# B&R Automation Studio project NAELD004C00R10L518F00 (part 15)

#### Act_OptP0937FBCtrl.st
```iecst
ACTION Act_OptP0937FBCtrl:

	fbJogSlowToFastDlyTm.PT			:= T#2s;
	fbJogSlowToFastDlyTm;
	fbLmtRstTm;

	//Conveyor Sensor Interruption
	IF p_tyDI.bPullerRetRS = FALSE AND eCurrPage = UIP0937AWPushOrPuller THEN
		tyP0937AWPushOrPuller.tyMotionStd.tyBtnStop.bRtCompl	:= TRUE;
	END_IF

//	IF EDGEPOS((p_udiAWPushOrPullerAxisErrID = 21570 OR p_udiAWPushOrPullerAxisErrID = 21571)
	IF EDGEPOS ((p_bAWPushOrPullerFwdLmtSen OR p_bAWPushOrPullerRevLmtSen)
		AND tyP0937AWPushOrPuller.tyMotionStd.tyBtnJogOpen.bValue = FALSE
		AND tyP0937AWPushOrPuller.tyMotionStd.tyBtnJogClose.bValue = FALSE)
	THEN
		fbLmtRstTm.IN	:= TRUE;
	END_IF

	IF fbLmtRstTm.Q = TRUE THEN
		tyP0937AWPushOrPuller.tyMotionStd.tyBtnRst.bRtCompl		:= TRUE;
	END_IF

	IF (tyP0937AWPushOrPuller.tyMotionStd.tyBtnJogOpen.bValue = FALSE AND tyP0937AWPushOrPuller.tyMotionStd.tyBtnJogClose.bValue = FALSE) AND (p_bAWPushOrPullerJogging = TRUE) THEN
		bJogStopAWPushOrPuller	:= TRUE;
	END_IF

	IF tyP0937AWPushOrPuller.tyMotionStd.tyBtnStop.bRtCompl = TRUE THEN
		eAWPushOrPullerAct		:= AWActStop;

		IF p_eAWPushOrPullerStat = AWActStop AND p_eAWPushOrPullerStatus = Done THEN
			eAWPushOrPullerAct	:= AWActIdle;

			tyP0937AWPushOrPuller.tyMotionStd.tyBtnStop.bRtCompl	:= FALSE;
			tyP0937AWPushOrPuller.tyMotionStd.tyBtnJogOpen.bRtCompl	:= FALSE;
			tyP0937AWPushOrPuller.tyMotionStd.tyBtnJogClose.bRtCompl:= FALSE;
			tyP0937AWPushOrPuller.tyMotionStd.tyBtnOrigin.bRtCompl	:= FALSE;
			tyP0937AWPushOrPuller.tyMotionStd.tyBtnMovAbs.bRtCompl	:= FALSE;
			tyP0937AWPushOrPuller.tyMotionStd.tyBtnMovRel.bRtCompl	:= FALSE;
			tyP0937AWPushOrPuller.tyAW.tyBtnGo.bRtCompl				:= FALSE;

			tyP0937AWPushOrPuller.tyMotionStd.tyBtnStop.bValue		:= TRUE;
			tyP0937AWPushOrPuller.tyMotionStd.tyBtnJogOpen.bValue	:= FALSE;
			tyP0937AWPushOrPuller.tyMotionStd.tyBtnJogClose.bValue	:= FALSE;
			tyP0937AWPushOrPuller.tyMotionStd.tyBtnOrigin.bValue	:= FALSE;
			tyP0937AWPushOrPuller.tyMotionStd.tyBtnMovAbs.bValue	:= FALSE;
			tyP0937AWPushOrPuller.tyMotionStd.tyBtnMovRel.bValue	:= FALSE;
			tyP0937AWPushOrPuller.tyAW.tyBtnGo.bValue				:= FALSE;

			tyP0937AWPushOrPuller.tyMotionStd.tyBtnStop.bRtLk		:= TRUE;
			tyP0937AWPushOrPuller.tyMotionStd.tyBtnJogOpen.bRtLk	:= FALSE;
			tyP0937AWPushOrPuller.tyMotionStd.tyBtnJogClose.bRtLk	:= FALSE;
			tyP0937AWPushOrPuller.tyMotionStd.tyBtnOrigin.bRtLk		:= FALSE;
			tyP0937AWPushOrPuller.tyMotionStd.tyBtnMovAbs.bRtLk		:= FALSE;
			tyP0937AWPushOrPuller.tyMotionStd.tyBtnMovRel.bRtLk		:= FALSE;
			tyP0937AWPushOrPuller.tyAW.tyBtnGo.bRtLk				:= FALSE;
		END_IF

	ELSIF (tyP0937AWPushOrPuller.tyMotionStd.tyBtnJogOpen.bRtCompl = TRUE) OR (tyP0937AWPushOrPuller.tyMotionStd.tyBtnJogClose.bRtCompl = TRUE) OR (bJogStopAWPushOrPuller = TRUE) THEN
		bJogSlow					:= FALSE;
		bJogFast					:= FALSE;
		fbJogSlowToFastDlyTm.IN		:= FALSE;

		eAWPushOrPullerAct		:= AWActJogStop;

		IF p_eAWPushOrPullerStat = AWActJogStop AND p_eAWPushOrPullerStatus = Done THEN
			eAWPushOrPullerAct	:= AWActIdle;

			bJogStopAWPushOrPuller	:= FALSE;

			tyP0937AWPushOrPuller.tyMotionStd.tyBtnStop.bRtCompl	:= FALSE;
			tyP0937AWPushOrPuller.tyMotionStd.tyBtnJogOpen.bRtCompl	:= FALSE;
			tyP0937AWPushOrPuller.tyMotionStd.tyBtnJogClose.bRtCompl:= FALSE;
			tyP0937AWPushOrPuller.tyMotionStd.tyBtnOrigin.bRtCompl	:= FALSE;
			tyP0937AWPushOrPuller.tyMotionStd.tyBtnMovAbs.bRtCompl	:= FALSE;
			tyP0937AWPushOrPuller.tyMotionStd.tyBtnMovRel.bRtCompl	:= FALSE;
			tyP0937AWPushOrPuller.tyAW.tyBtnGo.bRtCompl				:= FALSE;

			tyP0937AWPushOrPuller.tyMotionStd.tyBtnStop.bValue		:= TRUE;
			tyP0937AWPushOrPuller.tyMotionStd.tyBtnJogOpen.bValue	:= FALSE;
			tyP0937AWPushOrPuller.tyMotionStd.tyBtnJogClose.bValue	:= FALSE;
			tyP0937AWPushOrPuller.tyMotionStd.tyBtnOrigin.bValue	:= FALSE;
			tyP0937AWPushOrPuller.tyMotionStd.tyBtnMovAbs.bValue	:= FALSE;
			tyP0937AWPushOrPuller.tyMotionStd.tyBtnMovRel.bValue	:= FALSE;
			tyP0937AWPushOrPuller.tyAW.tyBtnGo.bValue				:= FALSE;

			tyP0937AWPushOrPuller.tyMotionStd.tyBtnStop.bRtLk		:= TRUE;
			tyP0937AWPushOrPuller.tyMotionStd.tyBtnJogOpen.bRtLk	:= FALSE;
			tyP0937AWPushOrPuller.tyMotionStd.tyBtnJogClose.bRtLk	:= FALSE;
			tyP0937AWPushOrPuller.tyMotionStd.tyBtnOrigin.bRtLk		:= FALSE;
			tyP0937AWPushOrPuller.tyMotionStd.tyBtnMovAbs.bRtLk		:= FALSE;
			tyP0937AWPushOrPuller.tyMotionStd.tyBtnMovRel.bRtLk		:= FALSE;
			tyP0937AWPushOrPuller.tyAW.tyBtnGo.bRtLk				:= FALSE;
		END_IF

	ELSIF tyP0937AWPushOrPuller.tyMotionStd.tyBtnPwr.bRtCompl = TRUE THEN
		tyP0937AWPushOrPuller.tyMotionStd.tyBtnPwr.bRtLk	:= TRUE;

		IF tyP0937AWPushOrPuller.tyMotionStd.tyBtnPwr.bValue = TRUE THEN
			eAWPushOrPullerAct		:= AWActPwrOn;

			IF p_eAWPushOrPullerStat = AWActPwrOn AND p_eAWPushOrPullerStatus = Done THEN
				eAWPushOrPullerAct	:= AWActIdle;

				tyP0937AWPushOrPuller.tyMotionStd.tyBtnPwr.bRtCompl	:= FALSE;
				tyP0937AWPushOrPuller.tyMotionStd.tyBtnPwr.bRtLk		:= FALSE;
			END_IF
		ELSE
			eAWPushOrPullerAct	:= AWActPwrOff;

			IF p_eAWPushOrPullerStat = AWActPwrOff AND p_eAWPushOrPullerStatus = Done THEN
				eAWPushOrPullerAct	:= AWActIdle;

				tyP0937AWPushOrPuller.tyMotionStd.tyBtnPwr.bRtCompl			:= FALSE;
				tyP0937AWPushOrPuller.tyMotionStd.tyBtnPwr.bRtLk			:= FALSE;
			END_IF
		END_IF

	ELSIF tyP0937AWPushOrPuller.tyMotionStd.tyBtnOrigin.bRtCompl = TRUE THEN
		tyP0937AWPushOrPuller.tyMotionStd.tyBtnOrigin.bValue	:= TRUE;
		tyP0937AWPushOrPuller.tyMotionStd.tyBtnStop.bValue	:= FALSE;

		tyP0937AWPushOrPuller.tyMotionStd.tyBtnOrigin.bRtLk	:= TRUE;
		tyP0937AWPushOrPuller.tyMotionStd.tyBtnStop.bRtLk		:= FALSE;

		eAWPushOrPullerAct		:= AWActHoming;

		IF p_eAWPushOrPullerStat = AWActHoming AND p_eAWPushOrPullerStatus = Done THEN
			eAWPushOrPullerAct	:= AWActIdle;

			tyP0937AWPushOrPuller.tyMotionStd.tyBtnOrigin.bRtCompl	:= FALSE;
			tyP0937AWPushOrPuller.tyMotionStd.tyBtnOrigin.bValue		:= FALSE;
			tyP0937AWPushOrPuller.tyMotionStd.tyBtnStop.bValue		:= TRUE;

			tyP0937AWPushOrPuller.tyMotionStd.tyBtnOrigin.bRtLk		:= FALSE;
			tyP0937AWPushOrPuller.tyMotionStd.tyBtnStop.bRtLk			:= TRUE;
		END_IF

	ELSIF tyP0937AWPushOrPuller.tyMotionStd.tyBtnRst.bRtCompl = TRUE THEN
		tyP0937AWPushOrPuller.tyMotionStd.tyBtnRst.bValue					:= TRUE;
		tyP0937AWPushOrPuller.tyMotionStd.tyBtnRst.bRtLk					:= TRUE;

		eAWPushOrPullerAct		:= AWActRstAxisErr;

		IF p_eAWPushOrPullerStat = AWActRstAxisErr AND p_eAWPushOrPullerStatus = Done THEN
			eAWPushOrPullerAct	:= AWActIdle;

			tyP0937AWPushOrPuller.tyMotionStd.tyBtnRst.bRtCompl		:= FALSE;
			tyP0937AWPushOrPuller.tyMotionStd.tyBtnRst.bValue			:= FALSE;
			tyP0937AWPushOrPuller.tyMotionStd.tyBtnRst.bRtLk			:= FALSE;

			fbLmtRstTm.IN			:= FALSE;
		END_IF

	ELSIF tyP0937AWPushOrPuller.tyAW.tyBtnGo.bRtCompl = TRUE THEN
		tyP0937AWPushOrPuller.tyAW.tyBtnGo.bValue				:= TRUE;
		tyP0937AWPushOrPuller.tyMotionStd.tyBtnStop.bValue	:= FALSE;

		tyP0937AWPushOrPuller.tyAW.tyBtnGo.bRtLk				:= TRUE;
		tyP0937AWPushOrPuller.tyMotionStd.tyBtnStop.bRtLk		:= FALSE;

		diMnlAWPushOrPullerGoWidth	:= (tyP0937AWPushOrPuller.tyAW.tyNumNewWidth.diValue)*3/4;
		diMnlAWPushOrPullerNomSpd		:= tyP0937AWPushOrPuller.tyMotionStd.tyNumNomSpd.diValue;

		eAWPushOrPullerAct		:= AWActGoWidth;

		IF p_eAWPushOrPullerStat = AWActGoWidth AND p_eAWPushOrPullerStatus = Done THEN
			eAWPushOrPullerAct	:= AWActIdle;

			tyP0937AWPushOrPuller.tyAW.tyBtnGo.bRtCompl			:= FALSE;
			tyP0937AWPushOrPuller.tyAW.tyBtnGo.bValue				:= FALSE;
			tyP0937AWPushOrPuller.tyMotionStd.tyBtnStop.bValue	:= TRUE;

			tyP0937AWPushOrPuller.tyAW.tyBtnGo.bRtLk				:= FALSE;
			tyP0937AWPushOrPuller.tyMotionStd.tyBtnStop.bRtLk		:= TRUE;
		END_IF

	ELSIF tyP0937AWPushOrPuller.tyMotionStd.tyBtnMovAbs.bRtCompl = TRUE THEN
		tyP0937AWPushOrPuller.tyMotionStd.tyBtnMovAbs.bValue		:= TRUE;
		tyP0937AWPushOrPuller.tyMotionStd.tyBtnStop.bValue		:= FALSE;

		tyP0937AWPushOrPuller.tyMotionStd.tyBtnMovAbs.bRtLk		:= TRUE;
		tyP0937AWPushOrPuller.tyMotionStd.tyBtnStop.bRtLk			:= FALSE;

		diMnlAWPushOrPullerTargetPos	:= tyP0937AWPushOrPuller.tyMotionStd.tyNumTargetPos.diValue;
		diMnlAWPushOrPullerNomSpd		:= tyP0937AWPushOrPuller.tyMotionStd.tyNumNomSpd.diValue;

		eAWPushOrPullerAct		:= AWActMovAbs;

		IF p_eAWPushOrPullerStat = AWActMovAbs AND p_eAWPushOrPullerStatus = Done THEN
			eAWPushOrPullerAct	:= AWActIdle;

			tyP0937AWPushOrPuller.tyMotionStd.tyBtnMovAbs.bRtCompl	:= FALSE;
			tyP0937AWPushOrPuller.tyMotionStd.tyBtnMovAbs.bValue		:= FALSE;
			tyP0937AWPushOrPuller.tyMotionStd.tyBtnStop.bValue		:= TRUE;

			tyP0937AWPushOrPuller.tyMotionStd.tyBtnMovAbs.bRtLk		:= FALSE;
			tyP0937AWPushOrPuller.tyMotionStd.tyBtnStop.bRtLk			:= TRUE;
		END_IF

	ELSIF tyP0937AWPushOrPuller.tyMotionStd.tyBtnMovRel.bRtCompl = TRUE THEN
		tyP0937AWPushOrPuller.tyMotionStd.tyBtnMovRel.bValue			:= TRUE;
		tyP0937AWPushOrPuller.tyMotionStd.tyBtnStop.bValue			:= FALSE;

		tyP0937AWPushOrPuller.tyMotionStd.tyBtnMovRel.bRtLk			:= TRUE;
		tyP0937AWPushOrPuller.tyMotionStd.tyBtnStop.bRtLk				:= FALSE;

		diMnlAWPushOrPullerStepSize	:= tyP0937AWPushOrPuller.tyMotionStd.tyNumStepSize.diValue;
		diMnlAWPushOrPullerNomSpd		:= tyP0937AWPushOrPuller.tyMotionStd.tyNumNomSpd.diValue;

		eAWPushOrPullerAct		:= AWActMovRel;

		IF p_eAWPushOrPullerStat = AWActMovRel AND p_eAWPushOrPullerStatus = Done THEN
			eAWPushOrPullerAct	:= AWActIdle;

			tyP0937AWPushOrPuller.tyMotionStd.tyBtnMovRel.bRtCompl	:= FALSE;
			tyP0937AWPushOrPuller.tyMotionStd.tyBtnMovRel.bValue		:= FALSE;
			tyP0937AWPushOrPuller.tyMotionStd.tyBtnStop.bValue		:= TRUE;

			tyP0937AWPushOrPuller.tyMotionStd.tyBtnMovRel.bRtLk		:= FALSE;
			tyP0937AWPushOrPuller.tyMotionStd.tyBtnStop.bRtLk			:= TRUE;
		END_IF

	ELSIF (tyP0937AWPushOrPuller.tyMotionStd.tyBtnJogOpen.bValue = TRUE) AND (fbJogSlowToFastDlyTm.Q = FALSE) AND (bJogSlow = FALSE) THEN
		tyP0937AWPushOrPuller.tyMotionStd.tyBtnStop.bValue		:= FALSE;
		tyP0937AWPushOrPuller.tyMotionStd.tyBtnStop.bRtLk			:= FALSE;

		fbJogSlowToFastDlyTm.IN	:= TRUE;

		diMnlAWPushOrPullerJogSpd		:= tyP0937AWPushOrPuller.tyMotionStd.tyNumSlwSpd.diValue;

		eAWPushOrPullerAct		:= AWActJogOpen;

		IF p_eAWPushOrPullerStat = AWActJogOpen AND p_eAWPushOrPullerStatus = Done THEN
			eAWPushOrPullerAct	:= AWActIdle;
			bJogSlow		:= TRUE;
		ELSIF p_eAWPushOrPullerStatus = Error THEN
			fbJogSlowToFastDlyTm.IN	:= FALSE;
			bJogSlow		:= TRUE;
		END_IF

	ELSIF (tyP0937AWPushOrPuller.tyMotionStd.tyBtnJogOpen.bValue = TRUE) AND (fbJogSlowToFastDlyTm.Q = TRUE) AND (bJogFast = FALSE) THEN
		tyP0937AWPushOrPuller.tyMotionStd.tyBtnStop.bValue	:= FALSE;
		tyP0937AWPushOrPuller.tyMotionStd.tyBtnStop.bRtLk		:= FALSE;

		fbJogSlowToFastDlyTm.IN		:= TRUE;

		diMnlAWPushOrPullerJogSpd		:= tyP0937AWPushOrPuller.tyMotionStd.tyNumNomSpd.diValue;

		eAWPushOrPullerAct	:= AWActJogOpen;

		IF p_eAWPushOrPullerStat = AWActJogOpen AND p_eAWPushOrPullerStatus = Done THEN
			eAWPushOrPullerAct	:= AWActIdle;
			bJogFast				:= TRUE;
		ELSIF p_eAWPushOrPullerStatus = Error THEN
			fbJogSlowToFastDlyTm.IN	:= FALSE;
			bJogFast				:= TRUE;
		END_IF

	ELSIF (tyP0937AWPushOrPuller.tyMotionStd.tyBtnJogClose.bValue = TRUE) AND (fbJogSlowToFastDlyTm.Q = FALSE) AND (bJogSlow = FALSE) THEN
		tyP0937AWPushOrPuller.tyMotionStd.tyBtnStop.bValue					:= FALSE;
		tyP0937AWPushOrPuller.tyMotionStd.tyBtnStop.bRtLk					:= FALSE;

		fbJogSlowToFastDlyTm.IN		:= TRUE;

		diMnlAWPushOrPullerJogSpd		:= tyP0937AWPushOrPuller.tyMotionStd.tyNumSlwSpd.diValue;

		eAWPushOrPullerAct		:= AWActJogClose;

		IF p_eAWPushOrPullerStat = AWActJogClose AND p_eAWPushOrPullerStatus = Done THEN
			eAWPushOrPullerAct	:= AWActIdle;
			bJogSlow				:= TRUE;
		ELSIF p_eAWPushOrPullerStatus = Error THEN
			fbJogSlowToFastDlyTm.IN	:= FALSE;
			bJogSlow				:= TRUE;
		END_IF

	ELSIF (tyP0937AWPushOrPuller.tyMotionStd.tyBtnJogClose.bValue = TRUE) AND (fbJogSlowToFastDlyTm.Q = TRUE) AND (bJogFast = FALSE) THEN
		tyP0937AWPushOrPuller.tyMotionStd.tyBtnStop.bValue	:= FALSE;
		tyP0937AWPushOrPuller.tyMotionStd.tyBtnStop.bRtLk		:= FALSE;

		fbJogSlowToFastDlyTm.IN		:= TRUE;

		diMnlAWPushOrPullerJogSpd		:= tyP0937AWPushOrPuller.tyMotionStd.tyNumNomSpd.diValue;

		eAWPushOrPullerAct			:= AWActJogClose;

		IF p_eAWPushOrPullerStat = AWActJogClose AND p_eAWPushOrPullerStatus = Done THEN
			eAWPushOrPullerAct	:= AWActIdle;
			bJogFast				:= TRUE;
		ELSIF p_eAWPushOrPullerStatus = Error THEN
			fbJogSlowToFastDlyTm.IN	:= FALSE;
			bJogFast				:= TRUE;
		END_IF

	END_IF

END_ACTION
```

#### Act_OptP0937FullMask.st
```iecst
ACTION Act_OptP0937FullMask:

	IF eCurrPage = UIP0937AWPushOrPuller THEN

		IF p_tyDI.bEStopSig = FALSE THEN
			p_tyC0002FullMask ACCESS ADR(tyP0937AWPushOrPuller.tyFullMaskEStop);

		ELSIF p_tyDI.bCoverSWSig = FALSE THEN
			p_tyC0002FullMask ACCESS ADR(tyP0937AWPushOrPuller.tyFullMaskCWSig);

		ELSIF p_tyDI.bSafetyRlySig = FALSE THEN
			p_tyC0002FullMask ACCESS ADR(tyP0937AWPushOrPuller.tyFullMaskSafetyRly);

		ELSIF p_tyDI.bConvLftSen THEN
			p_tyC0002FullMask ACCESS ADR(tyP0937AWPushOrPuller.tyFullMaskLftSenInterrupt);

		ELSIF p_tyDI.bConvRgtSen THEN
			p_tyC0002FullMask ACCESS ADR(tyP0937AWPushOrPuller.tyFullMaskRgtSenInterrupt);

		ELSIF p_tyNtParamCurr.bProjInletShutPrep AND (p_tyDI.bInShutterCloseRS = FALSE
			OR (p_tyDI.bInShutterCloseRS2 = FALSE AND p_tyNtParamCurr.tyDISettings.diInShutterCloseRS2 > 0)
			OR (p_tyDI.bInShutterCloseRS3 = FALSE AND p_tyNtParamCurr.tyDISettings.diInShutterCloseRS3 > 0)) THEN
			IF p_tyNtParamCurr.bProjCurtainSenPrep THEN
				IF p_tyDI.bInShutterCloseRS = FALSE OR p_tyDI.bInShutterCloseRS2 = FALSE OR p_tyDI.bInShutterCloseRS3 = FALSE THEN
					p_tyC0002FullMask ACCESS ADR(tyP0937AWPushOrPuller.tyFullMaskInShutOpnInterrupt);
				END_IF
			ELSE
				IF p_tyDI.bInShutterCloseRS = FALSE THEN
					p_tyC0002FullMask ACCESS ADR(tyP0937AWPushOrPuller.tyFullMaskInShutOpnInterrupt);
				END_IF
			END_IF

	//	ELSIF p_tyNtParamCurr.bProjOutletShutPrep AND p_tyDI.bOutShutterCloseRS = FALSE AND p_McParamOutShutterDis = FALSE THEN
		ELSIF p_tyNtParamCurr.bProjOutletShutPrep AND p_tyDI.bOutShutterCloseRS = FALSE THEN
			p_tyC0002FullMask ACCESS ADR(tyP0937AWPushOrPuller.tyFullMaskOutShutOpnInterrupt);

		ELSIF  p_tyDI.bPullerRetRS = FALSE OR p_tyDI.bPullerRotHmRS = FALSE THEN
			p_tyC0002FullMask ACCESS ADR(tyP0937AWPushOrPuller.tyFullMaskPullerRetInterrupt);

		ELSE
			p_tyC0002FullMask ACCESS ADR(tyP0937AWPushOrPuller.tyFullMaskHide);

		END_IF

	END_IF

END_ACTION
```

#### Act_OptP0937UpdtDat.st
```iecst
ACTION Act_OptP0937UpdtDat:

	tyP0937AWPushOrPuller.tyMotionStd.tyNumCurrPos.diValue		:= p_diAWPushOrPullerActualPos;
	tyP0937AWPushOrPuller.tyMotionStd.tyNumErrCode.diValue		:= UDINT_TO_DINT(p_udiAWPushOrPullerAxisErrID);
	tyP0937AWPushOrPuller.tyMotionStd.tyBitmapPwr.usiValueIdx		:= BOOL_TO_USINT(p_bAWPushOrPullerPwrOn);
	tyP0937AWPushOrPuller.tyMotionStd.tyBitmapRst.usiValueIdx		:= BOOL_TO_USINT(NOT p_bAWPushOrPullerAxisErr);
	tyP0937AWPushOrPuller.tyMotionStd.tyBitmapOrigin.usiValueIdx	:= BOOL_TO_USINT(p_bAWPushOrPullerIsHomed);
	tyP0937AWPushOrPuller.tyMotionStd.tyBtnOpenLmtSen.bValue		:= p_bAWPushOrPullerCloseSen;
	tyP0937AWPushOrPuller.tyMotionStd.tyBtnCloseLmtSen.bValue		:= p_bAWPushOrPullerOpenSen;

	IF p_bAWPushOrPullerIsHomed = TRUE THEN
		IF p_diAWPushOrPullerActualPos <= (p_tyNtParamCurr.tyProdRcpWidth.diMax / 2) THEN
			tyP0937AWPushOrPuller.tyMotionStd.tyBitmapMc.uiValueIdx 	:= 38;
		ELSE
			tyP0937AWPushOrPuller.tyMotionStd.tyBitmapMc.uiValueIdx 	:= 39;
		END_IF
	ELSE
		tyP0937AWPushOrPuller.tyMotionStd.tyBitmapMc.uiValueIdx	:= 38;
	END_IF

	IF p_tyNtParamCurr.eProjMag = LDMagTriple AND p_tyNtParamCurr.bMagAutoVerifyPrep = FALSE AND p_tyNtParamCurr.bProjMotorizedPullerPrep = TRUE
		AND p_tyNtParamCurr.bProjCurtainSenPrep = FALSE THEN
		IF 	tyP0937AWPushOrPuller.tyMotionStd.tyBitmapMc.uiValueIdx < 300 THEN
			tyP0937AWPushOrPuller.tyMotionStd.tyBitmapMc.uiValueIdx	:= tyP0937AWPushOrPuller.tyMotionStd.tyBitmapMc.uiValueIdx + 300;
		END_IF
	ELSIF p_tyNtParamCurr.eProjMag = LDMagTriple AND p_tyNtParamCurr.bMagAutoVerifyPrep = FALSE AND p_tyNtParamCurr.bProjMotorizedPullerPrep = TRUE
		AND p_tyNtParamCurr.bProjCurtainSenPrep = TRUE AND p_tyNtParamCurr.bProjTopToBtmDefault = TRUE THEN
		IF 	tyP0937AWPushOrPuller.tyMotionStd.tyBitmapMc.uiValueIdx < 373-38 THEN
			tyP0937AWPushOrPuller.tyMotionStd.tyBitmapMc.uiValueIdx	:= tyP0937AWPushOrPuller.tyMotionStd.tyBitmapMc.uiValueIdx + 373-38;
		END_IF
	ELSIF p_tyNtParamCurr.eProjMag = LDMagTriple AND p_tyNtParamCurr.bMagAutoVerifyPrep = FALSE AND p_tyNtParamCurr.bProjMotorizedPullerPrep = TRUE
		AND p_tyNtParamCurr.bProjCurtainSenPrep = TRUE AND p_tyNtParamCurr.bProjTopToBtmDefault = FALSE THEN
		IF 	tyP0937AWPushOrPuller.tyMotionStd.tyBitmapMc.uiValueIdx < 428-38 THEN
			tyP0937AWPushOrPuller.tyMotionStd.tyBitmapMc.uiValueIdx	:= tyP0937AWPushOrPuller.tyMotionStd.tyBitmapMc.uiValueIdx + 428-38;

		END_IF
	END_IF

END_ACTION
```

#### Act_EntP0939Disp.st
```iecst
ACTION Act_EntP0939Disp:

	//Access Address
	p_tyC0002FullMask ACCESS ADR(tyP0939MagConv4.tyFullMaskHide);

//	p_tyC0004Navi ACCESS ADR(tyP0939MagConv4.tyNaviBack);
	p_tyC0004Navi ACCESS ADR(tyP0939MagConv4.tyNavi4Lyr4);

	p_tyC0005Main ACCESS ADR(tyCommon.tyMain);

	p_tyC0007Notif ACCESS ADR(tyCommon.tyNotif);

	p_tyC0008MsgBox ACCESS ADR(tyP0939MagConv4.tyMsgBoxHide);

	p_tyC0009Info ACCESS ADR(tyCommon.tyInfo);

	p_tyP0939Mag4ConvCom ACCESS ADR(tyP0939MagConv4.tyCom);
	p_tyP0939Mag4ConvDC ACCESS ADR(tyP0939MagConv4.tyDC);
	p_tyP0939Mag4ConvFB ACCESS ADR(tyP0939MagConv4.tyFB);

	IF p_tyNtParamCurr.eProjMag = LDMagDual AND p_tyNtParamCurr.bMagAutoVerifyPrep = FALSE THEN
		tyP0939MagConv4.tyCom.tyBitmapMc.usiValueIdx	:= 111;
	ELSIF p_tyNtParamCurr.eProjMag = LDMagDual AND p_tyNtParamCurr.bMagAutoVerifyPrep = TRUE THEN
		tyP0939MagConv4.tyCom.tyBitmapMc.usiValueIdx	:= 200;
	ELSIF p_tyNtParamCurr.eProjMag = LDMagTriple AND p_tyNtParamCurr.bMagAutoVerifyPrep = TRUE THEN
		tyP0939MagConv4.tyCom.tyBitmapMc.usiValueIdx	:= 0;
	ELSIF p_tyNtParamCurr.eProjMag = LDMagQuadruple AND p_tyNtParamCurr.bMagAutoVerifyPrep = TRUE THEN
		tyP0939MagConv4.tyCom.tyBitmapMc.usiValueIdx	:= 116;
	ELSE
		tyP0939MagConv4.tyCom.tyBitmapMc.usiValueIdx	:= 100;
	END_IF

	IF p_tyNtParamCurr.bMagAutoVerifyPrep = FALSE THEN
		tyP0939MagConv4.tyFB.tyBtnFixedClamp.usiTxtIdx	:= 6;
		tyP0939MagConv4.tyFB.tyBtnFixedUnclamp.usiTxtIdx:= 6;
		tyP0939MagConv4.tyFB.tyBtnRemoteClamp.usiTxtIdx	:= 6;
		tyP0939MagConv4.tyFB.tyBtnRemoteUnclamp.usiTxtIdx:= 6;
	ELSE
		tyP0939MagConv4.tyFB.tyBtnFixedClamp.usiTxtIdx	:= 6;
		tyP0939MagConv4.tyFB.tyBtnFixedUnclamp.usiTxtIdx:= 6;
		tyP0939MagConv4.tyFB.tyBtnRemoteClamp.usiTxtIdx	:= 6;
		tyP0939MagConv4.tyFB.tyBtnRemoteUnclamp.usiTxtIdx:= 6;

	END_IF

	IF p_tyNtParamCurr.bMagAutoVerifyPrep = FALSE THEN
		IF tyP0939MagConv4.tyCom.tyBtnSwitch.bValue THEN
			fUIInRtStatHide(ADR(tyP0939MagConv4.tyFB.tyLyr.uiRtStat));
			fUIInRtStatHide(ADR(tyP0939MagConv4.tyDC.tyLyr.uiRtStat));
			fUIInRtStatHide(ADR(tyP0939MagConv4.tyFB.tyLyrWithoutSelClamp.uiRtStat));
			fUIInRtStatOff(ADR(tyP0939MagConv4.tyDC.tyLyrWithoutSelClamp.uiRtStat));
		ELSE
			fUIInRtStatHide(ADR(tyP0939MagConv4.tyFB.tyLyr.uiRtStat));
			fUIInRtStatHide(ADR(tyP0939MagConv4.tyDC.tyLyr.uiRtStat));
			fUIInRtStatOff(ADR(tyP0939MagConv4.tyFB.tyLyrWithoutSelClamp.uiRtStat));
			fUIInRtStatHide(ADR(tyP0939MagConv4.tyDC.tyLyrWithoutSelClamp.uiRtStat));
		END_IF
	ELSE
		IF tyP0939MagConv4.tyCom.tyBtnSwitch.bValue THEN
			fUIInRtStatHide(ADR(tyP0939MagConv4.tyFB.tyLyr.uiRtStat));
			fUIInRtStatOff(ADR(tyP0939MagConv4.tyDC.tyLyr.uiRtStat));
			fUIInRtStatHide(ADR(tyP0939MagConv4.tyFB.tyLyrWithoutSelClamp.uiRtStat));
			fUIInRtStatHide(ADR(tyP0939MagConv4.tyDC.tyLyrWithoutSelClamp.uiRtStat));
		ELSE
			fUIInRtStatOff(ADR(tyP0939MagConv4.tyFB.tyLyr.uiRtStat));
			fUIInRtStatHide(ADR(tyP0939MagConv4.tyDC.tyLyr.uiRtStat));
			fUIInRtStatHide(ADR(tyP0939MagConv4.tyFB.tyLyrWithoutSelClamp.uiRtStat));
			fUIInRtStatHide(ADR(tyP0939MagConv4.tyDC.tyLyrWithoutSelClamp.uiRtStat));
		END_IF
	END_IF

END_ACTION
```

#### Act_OptP0939FullMask.st
```iecst
ACTION Act_OptP0939FullMask:

	IF eCurrPage = UIP0939MagConv4 THEN

		IF p_tyDI.bEStopSig = FALSE THEN
			p_tyC0002FullMask ACCESS ADR(tyP0939MagConv4.tyFullMaskEStop);

		ELSIF p_tyDI.bCoverSWSig = FALSE THEN
			p_tyC0002FullMask ACCESS ADR(tyP0939MagConv4.tyFullMaskCWSig);

		ELSIF p_tyDI.bSafetyRlySig = FALSE THEN
			p_tyC0002FullMask ACCESS ADR(tyP0939MagConv4.tyFullMaskSafetyRly);

		ELSE
			p_tyC0002FullMask ACCESS ADR(tyP0939MagConv4.tyFullMaskHide);

		END_IF

	END_IF

END_ACTION
```

#### Act_OptP0939Navi.st
```iecst
ACTION Act_OptP0939Navi:

	IF tyP0939MagConv4.tyNavi4Lyr4.tyBtnBack.bRtCompl = TRUE THEN
		tyP0939MagConv4.tyNavi4Lyr4.tyBtnBack.bRtCompl	:= FALSE;
		tyP0939MagConv4.tyNavi4Lyr4.tyBtnBack.bValue	:= FALSE;

		eChgPage	:= UIP0920MtrNPneuCtrl;

		bDispMagConv1	:= FALSE;
		bDispMagConv2	:= FALSE;
		bDispMagConv3	:= FALSE;
		bDispMagConv4	:= TRUE;

	ELSIF tyP0939MagConv4.tyNavi4Lyr4.tyBtnLeft.bRtCompl = TRUE THEN
		tyP0939MagConv4.tyNavi4Lyr4.tyBtnLeft.bRtCompl			:= FALSE;
		tyP0939MagConv4.tyNavi4Lyr4.tyBtnLeft.bValue			:= FALSE;
		eChgPage												:= UIP0932MagConv3;
		bDispMagConv1	:= FALSE;
		bDispMagConv2	:= FALSE;
		bDispMagConv3	:= TRUE;
		bDispMagConv4	:= FALSE;

	ELSIF tyP0939MagConv4.tyNavi4Lyr4.tyBtnRgt.bRtCompl = TRUE THEN
		tyP0939MagConv4.tyNavi4Lyr4.tyBtnRgt.bRtCompl			:= FALSE;
		tyP0939MagConv4.tyNavi4Lyr4.tyBtnRgt.bValue				:= FALSE;
		eChgPage												:= UIP0930MagConv1;
		bDispMagConv1	:= TRUE;
		bDispMagConv2	:= FALSE;
		bDispMagConv3	:= FALSE;
		bDispMagConv4	:= FALSE;

	END_IF

END_ACTION
```

#### Act_OptP0939MagConv4ChgLyr.st
```iecst
ACTION Act_OptP0939MagConv4ChgLyr:

	IF p_tyNtParamCurr.bMagAutoVerifyPrep THEN
		IF tyP0939MagConv4.tyCom.tyBtnSwitch.bRtCompl THEN
			tyP0939MagConv4.tyCom.tyBtnSwitch.bRtCompl	:= FALSE;

			IF tyP0939MagConv4.tyCom.tyBtnSwitch.bValue = TRUE THEN
				fUIInRtStatOff(ADR(tyP0939MagConv4.tyDC.tyLyr.uiRtStat));
				fUIInRtStatHide(ADR(tyP0939MagConv4.tyFB.tyLyr.uiRtStat));
			ELSE
				fUIInRtStatHide(ADR(tyP0939MagConv4.tyDC.tyLyr.uiRtStat));
				fUIInRtStatOff(ADR(tyP0939MagConv4.tyFB.tyLyr.uiRtStat));
			END_IF

		END_IF
	ELSE
		IF tyP0939MagConv4.tyCom.tyBtnSwitch.bRtCompl THEN
			tyP0939MagConv4.tyCom.tyBtnSwitch.bRtCompl	:= FALSE;

			IF tyP0939MagConv4.tyCom.tyBtnSwitch.bValue = TRUE THEN
				fUIInRtStatOff(ADR(tyP0939MagConv4.tyDC.tyLyrWithoutSelClamp.uiRtStat));
				fUIInRtStatHide(ADR(tyP0939MagConv4.tyFB.tyLyrWithoutSelClamp.uiRtStat));
			ELSE
				fUIInRtStatHide(ADR(tyP0939MagConv4.tyDC.tyLyrWithoutSelClamp.uiRtStat));
				fUIInRtStatOff(ADR(tyP0939MagConv4.tyFB.tyLyrWithoutSelClamp.uiRtStat));
			END_IF

		END_IF
	END_IF

END_ACTION
```

#### Act_OptP0939MagConv4Sen.st
```iecst
ACTION Act_OptP0939MagConv4Sen:

	tyP0939MagConv4.tyCom.tyBtnMagPresentSen.bValue			:= p_tyDI.bMagPresentSen4;
	tyP0939MagConv4.tyCom.tyBtnMagConvEntSen.bValue			:= p_tyDI.bMagConvEntSen4;
	tyP0939MagConv4.tyCom.tyBtnMagAIVPosSen1.bValue			:= p_tyDI.bMag4AGVInPosSen1;
	tyP0939MagConv4.tyCom.tyBtnMagAIVPosSen2.bValue			:= p_tyDI.bMag4AGVInPosSen2;
	tyP0939MagConv4.tyCom.tyBtnMagOrientationChkSen1.bValue	:= p_tyDI.bMag4OrientChkSen1;
	tyP0939MagConv4.tyCom.tyBtnMagOrientationChkSen2.bValue	:= p_tyDI.bMag4OrientChkSen2;

	tyP0939MagConv4.tyCom.tyBtnFixedClampRS.bValue			:= p_tyDI.bMag4FixedClampRS;
	tyP0939MagConv4.tyCom.tyBtnFixedUnclampRS.bValue		:= p_tyDI.bMag4FixedUnclampRS;
	tyP0939MagConv4.tyCom.tyBtnRemoteClampRS.bValue			:= p_tyDI.bMag4RemoteClampRS;
	tyP0939MagConv4.tyCom.tyBtnRemoteUnclampRS.bValue		:= p_tyDI.bMag4RemoteUnclampRS;

	tyP0939MagConv4.tyCom.tyBtnSelUnclampRS.bValue			:= p_tyDI.bMag4SelUnClampRS;

	tyP0939MagConv4.tyCom.tyBtnCAB717Sen.bValue				:= p_tyDI.bMagConvCAB717MagSen4;
	tyP0939MagConv4.tyCom.tyBtnHeightSen.bValue				:= p_tyDI.bMagConvHeightSen4;
	tyP0939MagConv4.tyCom.tyBtnMagSmallSen.bValue			:= p_tyDI.bMagConvSmallMagSen4;
	tyP0939MagConv4.tyCom.tyBtnMagLargeSen.bValue			:= p_tyDI.bMagConvLargeMagSen4;

	//Machine Bitmap
	IF p_tyNtParamCurr.bMagAutoVerifyPrep = FALSE THEN
		IF tyP0939MagConv4.tyFB.tyBtnFixedClamp.bRtCompl OR  tyP0939MagConv4.tyFB.tyBtnRemoteClamp.bRtCompl
			OR tyP0939MagConv4.tyDC.tyBtnFixedClamp.bRtCompl OR tyP0939MagConv4.tyDC.tyBtnRemoteClamp.bRtCompl  THEN

			tyP0939MagConv4.tyCom.tyBitmapMc.usiValueIdx	:= 2;

		ELSIF tyP0939MagConv4.tyFB.tyBtnFixedUnclamp.bRtCompl OR tyP0939MagConv4.tyFB.tyBtnRemoteUnclamp.bRtCompl
			OR tyP0939MagConv4.tyDC.tyBtnFixedUnclamp.bRtCompl OR tyP0939MagConv4.tyDC.tyBtnRemoteUnclamp.bRtCompl  THEN

			tyP0939MagConv4.tyCom.tyBitmapMc.usiValueIdx	:= 1;

		ELSIF tyP0939MagConv4.tyFB.tyBtnEnt.bRtCompl OR tyP0939MagConv4.tyFB.tyBtnExit.bRtCompl OR tyP0939MagConv4.tyFB.tyBtnStop.bRtCompl
			OR tyP0939MagConv4.tyDC.tyBtnMagIn.bRtCompl OR tyP0939MagConv4.tyDC.tyBtnMagOut.bRtCompl OR tyP0939MagConv4.tyDC.tyBtnStop.bRtCompl THEN

			tyP0939MagConv4.tyCom.tyBitmapMc.usiValueIdx	:= 0;

		END_IF

	ELSIF p_tyNtParamCurr.eProjMag = LDMagTriple AND p_tyNtParamCurr.bMagAutoVerifyPrep THEN
		IF tyP0939MagConv4.tyFB.tyBtnFixedClamp.bRtCompl
			OR tyP0939MagConv4.tyDC.tyBtnFixedClamp.bRtCompl THEN

			tyP0939MagConv4.tyCom.tyBitmapMc.usiValueIdx	:= 2;

		ELSIF tyP0939MagConv4.tyFB.tyBtnFixedUnclamp.bRtCompl
			OR tyP0939MagConv4.tyDC.tyBtnFixedUnclamp.bRtCompl THEN

			tyP0939MagConv4.tyCom.tyBitmapMc.usiValueIdx	:= 1;

		ELSIF tyP0939MagConv4.tyFB.tyBtnRemoteClamp.bRtCompl
			OR tyP0939MagConv4.tyDC.tyBtnRemoteClamp.bRtCompl THEN

			tyP0939MagConv4.tyCom.tyBitmapMc.usiValueIdx	:= 14;

		ELSIF tyP0939MagConv4.tyFB.tyBtnRemoteUnclamp.bRtCompl
			OR tyP0939MagConv4.tyDC.tyBtnRemoteUnclamp.bRtCompl THEN

			tyP0939MagConv4.tyCom.tyBitmapMc.usiValueIdx	:= 13;

		ELSIF tyP0939MagConv4.tyFB.tyBtnSelClamp.bRtCompl
			OR tyP0939MagConv4.tyDC.tyBtnSelClamp.bRtCompl THEN

			tyP0939MagConv4.tyCom.tyBitmapMc.usiValueIdx	:= 20;

		ELSIF tyP0939MagConv4.tyFB.tyBtnSelUnclamp.bRtCompl
			OR tyP0939MagConv4.tyDC.tyBtnSelUnclamp.bRtCompl THEN

			tyP0939MagConv4.tyCom.tyBitmapMc.usiValueIdx	:= 19;

		ELSIF tyP0939MagConv4.tyFB.tyBtnEnt.bRtCompl OR tyP0939MagConv4.tyFB.tyBtnExit.bRtCompl OR tyP0939MagConv4.tyFB.tyBtnStop.bRtCompl
			OR tyP0939MagConv4.tyDC.tyBtnMagIn.bRtCompl OR tyP0939MagConv4.tyDC.tyBtnMagOut.bRtCompl OR tyP0939MagConv4.tyDC.tyBtnStop.bRtCompl THEN

			tyP0939MagConv4.tyCom.tyBitmapMc.usiValueIdx	:= 0;

		END_IF

	ELSIF p_tyNtParamCurr.eProjMag = LDMagQuadruple AND p_tyNtParamCurr.bMagAutoVerifyPrep THEN
		IF tyP0939MagConv4.tyFB.tyBtnFixedClamp.bRtCompl
			OR tyP0939MagConv4.tyDC.tyBtnFixedClamp.bRtCompl THEN

			tyP0939MagConv4.tyCom.tyBitmapMc.usiValueIdx	:= 118;

		ELSIF tyP0939MagConv4.tyFB.tyBtnFixedUnclamp.bRtCompl
			OR tyP0939MagConv4.tyDC.tyBtnFixedUnclamp.bRtCompl THEN

			tyP0939MagConv4.tyCom.tyBitmapMc.usiValueIdx	:= 117;

		ELSIF tyP0939MagConv4.tyFB.tyBtnRemoteClamp.bRtCompl
			OR tyP0939MagConv4.tyDC.tyBtnRemoteClamp.bRtCompl THEN

			tyP0939MagConv4.tyCom.tyBitmapMc.usiValueIdx	:= 120;

		ELSIF tyP0939MagConv4.tyFB.tyBtnRemoteUnclamp.bRtCompl
			OR tyP0939MagConv4.tyDC.tyBtnRemoteUnclamp.bRtCompl THEN

			tyP0939MagConv4.tyCom.tyBitmapMc.usiValueIdx	:= 119;

		ELSIF tyP0939MagConv4.tyFB.tyBtnSelClamp.bRtCompl
			OR tyP0939MagConv4.tyDC.tyBtnSelClamp.bRtCompl THEN

			tyP0939MagConv4.tyCom.tyBitmapMc.usiValueIdx	:= 122;

		ELSIF tyP0939MagConv4.tyFB.tyBtnSelUnclamp.bRtCompl
			OR tyP0939MagConv4.tyDC.tyBtnSelUnclamp.bRtCompl THEN

			tyP0939MagConv4.tyCom.tyBitmapMc.usiValueIdx	:= 121;

		ELSIF tyP0939MagConv4.tyFB.tyBtnEnt.bRtCompl OR tyP0939MagConv4.tyFB.tyBtnExit.bRtCompl OR tyP0939MagConv4.tyFB.tyBtnStop.bRtCompl
			OR tyP0939MagConv4.tyDC.tyBtnMagIn.bRtCompl OR tyP0939MagConv4.tyDC.tyBtnMagOut.bRtCompl OR tyP0939MagConv4.tyDC.tyBtnStop.bRtCompl THEN

			tyP0939MagConv4.tyCom.tyBitmapMc.usiValueIdx	:= 116;

		END_IF
	END_IF

	IF p_tyNtParamCurr.eProjMag = LDMagTriple AND p_tyNtParamCurr.bMagAutoVerifyPrep = FALSE THEN
		IF tyP0939MagConv4.tyCom.tyBitmapMc.usiValueIdx < 100 THEN
			tyP0939MagConv4.tyCom.tyBitmapMc.usiValueIdx	:= tyP0939MagConv4.tyCom.tyBitmapMc.usiValueIdx + 100;
		END_IF
	ELSIF p_tyNtParamCurr.eProjMag = LDMagDual AND p_tyNtParamCurr.bMagAutoVerifyPrep = TRUE THEN
		IF tyP0939MagConv4.tyCom.tyBitmapMc.usiValueIdx < 200 THEN
			tyP0939MagConv4.tyCom.tyBitmapMc.usiValueIdx	:= tyP0939MagConv4.tyCom.tyBitmapMc.usiValueIdx + 200;
		END_IF

	END_IF

END_ACTION
```

#### Act_OptP0939MagConv4FB.st
```iecst
ACTION Act_OptP0939MagConv4FB:

	//Magazine Conveyor
	IF tyP0939MagConv4.tyFB.tyBtnStop.bRtCompl = TRUE THEN
		eMagConv2Clp4Act	:= MagConv2ClpActStop;

		IF p_eMagConv2Clp4Stat = MagConv2ClpActStop AND p_eMagConv2Clp4Status = Done THEN
			eMagConv2Clp4Act	:= MagConv2ClpActIdle;

			tyP0939MagConv4.tyFB.tyBtnEnt.bRtCompl	:= FALSE;
			tyP0939MagConv4.tyFB.tyBtnEnt.bValue	:= FALSE;
			tyP0939MagConv4.tyFB.tyBtnEnt.bRtLk		:= FALSE;

			tyP0939MagConv4.tyFB.tyBtnExit.bRtCompl	:= FALSE;
			tyP0939MagConv4.tyFB.tyBtnExit.bValue	:= FALSE;
			tyP0939MagConv4.tyFB.tyBtnExit.bRtLk	:= FALSE;

			tyP0939MagConv4.tyFB.tyBtnStop.bRtCompl	:= FALSE;
			tyP0939MagConv4.tyFB.tyBtnStop.bValue	:= TRUE;
			tyP0939MagConv4.tyFB.tyBtnStop.bRtLk	:= TRUE;
		END_IF

	ELSIF tyP0939MagConv4.tyFB.tyBtnEnt.bRtCompl = TRUE THEN
		tyP0939MagConv4.tyFB.tyBtnEnt.bValue	:= TRUE;
		tyP0939MagConv4.tyFB.tyBtnEnt.bRtLk		:= TRUE;

		tyP0939MagConv4.tyFB.tyBtnStop.bValue	:= FALSE;
		tyP0939MagConv4.tyFB.tyBtnStop.bRtLk	:= FALSE;

		eMagConv2Clp4Act	:= MagConv2ClpActEnt;

		IF p_eMagConv2Clp4Stat = MagConv2ClpActEnt AND p_eMagConv2Clp4Status = Done THEN
			eMagConv2Clp4Act	:= MagConv2ClpActIdle;

			tyP0939MagConv4.tyFB.tyBtnEnt.bRtCompl	:= FALSE;

			tyP0939MagConv4.tyFB.tyBtnEnt.bValue	:= FALSE;
			tyP0939MagConv4.tyFB.tyBtnEnt.bRtLk		:= FALSE;

			tyP0939MagConv4.tyFB.tyBtnStop.bValue	:= TRUE;
			tyP0939MagConv4.tyFB.tyBtnStop.bRtLk	:= TRUE;
		END_IF

	ELSIF (p_eMagConv2Clp4Stat = MagConv2ClpActPreExit AND p_eMagConv2Clp4Status = Done) THEN
		eMagConv2Clp4Act	:= MagConv2ClpActIdle;

		tyP0939MagConv4.tyFB.tyBtnExit.bRtCompl	:= FALSE;

		tyP0939MagConv4.tyFB.tyBtnExit.bValue	:= FALSE;
		tyP0939MagConv4.tyFB.tyBtnExit.bRtLk	:= FALSE;

		tyP0939MagConv4.tyFB.tyBtnStop.bValue	:= TRUE;
		tyP0939MagConv4.tyFB.tyBtnStop.bRtLk	:= TRUE;

	ELSIF (p_eMagConv2Clp4Stat = MagConv2ClpActExit AND p_eMagConv2Clp4Status = Done) THEN
		eMagConv2Clp4Act	:= MagConv2ClpActIdle;

		tyP0939MagConv4.tyFB.tyBtnExit.bRtCompl	:= FALSE;

		tyP0939MagConv4.tyFB.tyBtnExit.bValue	:= FALSE;
		tyP0939MagConv4.tyFB.tyBtnExit.bRtLk	:= FALSE;

		tyP0939MagConv4.tyFB.tyBtnStop.bValue	:= TRUE;
		tyP0939MagConv4.tyFB.tyBtnStop.bRtLk	:= TRUE;

	ELSIF tyP0939MagConv4.tyFB.tyBtnExit.bRtCompl = TRUE THEN
		tyP0939MagConv4.tyFB.tyBtnExit.bRtCompl	:= FALSE;
		tyP0939MagConv4.tyFB.tyBtnExit.bValue	:= TRUE;
		tyP0939MagConv4.tyFB.tyBtnExit.bRtLk	:= TRUE;

		tyP0939MagConv4.tyFB.tyBtnStop.bValue	:= FALSE;
		tyP0939MagConv4.tyFB.tyBtnStop.bRtLk	:= FALSE;

		IF p_tyDI.bMagConvEntSen4  THEN
			eMagConv2Clp4Act	:= MagConv2ClpActExit;
		ELSE
			IF p_tyDI.bMagPresentSen4 THEN
				eMagConv2Clp4Act	:= MagConv2ClpActPreExit;
			ELSE
				eMagConv2Clp4Act	:= MagConv2ClpActExit;
			END_IF
		END_IF
	END_IF

	//Magazine Clamper
	IF tyP0939MagConv4.tyCom.tyBtnSwitch.bValue = FALSE THEN

		//Fixed/Bottom
		IF tyP0939MagConv4.tyFB.tyBtnFixedUnclamp.bRtCompl = TRUE THEN
			tyP0939MagConv4.tyFB.tyBtnFixedUnclamp.bRtCompl	:= FALSE;

			tyP0939MagConv4.tyFB.tyBtnFixedUnclamp.bValue	:= TRUE;
			tyP0939MagConv4.tyFB.tyBtnFixedClamp.bValue		:= FALSE;

		ELSIF tyP0939MagConv4.tyFB.tyBtnFixedClamp.bRtCompl = TRUE THEN
			tyP0939MagConv4.tyFB.tyBtnFixedClamp.bRtCompl	:= FALSE;

			tyP0939MagConv4.tyFB.tyBtnFixedClamp.bValue		:= TRUE;
			tyP0939MagConv4.tyFB.tyBtnFixedUnclamp.bValue	:= FALSE;

		END_IF

		//Remote/Top
		IF tyP0939MagConv4.tyFB.tyBtnRemoteUnclamp.bRtCompl = TRUE THEN
			tyP0939MagConv4.tyFB.tyBtnRemoteUnclamp.bRtCompl	:= FALSE;

			tyP0939MagConv4.tyFB.tyBtnRemoteUnclamp.bValue	:= TRUE;
			tyP0939MagConv4.tyFB.tyBtnRemoteClamp.bValue	:= FALSE;

		ELSIF tyP0939MagConv4.tyFB.tyBtnRemoteClamp.bRtCompl = TRUE THEN
			tyP0939MagConv4.tyFB.tyBtnRemoteClamp.bRtCompl	:= FALSE;

			tyP0939MagConv4.tyFB.tyBtnRemoteClamp.bValue	:= TRUE;
			tyP0939MagConv4.tyFB.tyBtnRemoteUnclamp.bValue	:= FALSE;

		END_IF

		//Selection
		IF tyP0939MagConv4.tyFB.tyBtnSelUnclamp.bRtCompl = TRUE THEN
			tyP0939MagConv4.tyFB.tyBtnSelUnclamp.bRtCompl	:= FALSE;

			tyP0939MagConv4.tyFB.tyBtnSelUnclamp.bValue	:= TRUE;
			tyP0939MagConv4.tyFB.tyBtnSelClamp.bValue	:= FALSE;

		ELSIF tyP0939MagConv4.tyFB.tyBtnSelClamp.bRtCompl = TRUE THEN
			tyP0939MagConv4.tyFB.tyBtnSelClamp.bRtCompl	:= FALSE;

			tyP0939MagConv4.tyFB.tyBtnSelClamp.bValue	:= TRUE;
			tyP0939MagConv4.tyFB.tyBtnSelUnclamp.bValue	:= FALSE;

		END_IF

		// Fixed Clamper
		IF tyP0939MagConv4.tyFB.tyBtnFixedUnclamp.bValue = TRUE THEN

			eMagConv2Clp4Act	:= MagConv2ClpActFixClprUnclamp;

			IF p_eMagConv2Clp4Stat = MagConv2ClpActFixClprUnclamp AND p_eMagConv2Clp4Status = Done THEN

				eMagConv2Clp4Act	:= MagConv2ClpActIdle;

				tyP0939MagConv4.tyFB.tyBtnFixedUnclamp.bValue	:= FALSE;

			ELSIF p_eMagConv2Clp4Status = Error THEN

				tyP0939MagConv4.tyFB.tyBtnFixedUnclamp.bValue	:= FALSE;

			END_IF

		ELSIF tyP0939MagConv4.tyFB.tyBtnFixedClamp.bValue = TRUE THEN
			eMagConv2Clp4Act	:= MagConv2ClpActFixClprClamp;

			IF p_eMagConv2Clp4Stat = MagConv2ClpActFixClprClamp AND p_eMagConv2Clp4Status = Done THEN

				eMagConv2Clp4Act	:= MagConv2ClpActIdle;

				tyP0939MagConv4.tyFB.tyBtnFixedClamp.bValue := FALSE;

			ELSIF p_eMagConv2Clp4Status = Error THEN

				tyP0939MagConv4.tyFB.tyBtnFixedClamp.bValue := FALSE;

			END_IF

		END_IF

		//Remote Clamper
		IF tyP0939MagConv4.tyFB.tyBtnRemoteUnclamp.bValue = TRUE THEN

			eMagConv2Clp4Act	:= MagConv2ClpActRmtClprUnclamp;

			IF p_eMagConv2Clp4Stat = MagConv2ClpActRmtClprUnclamp AND p_eMagConv2Clp4Status = Done THEN

				eMagConv2Clp4Act	:= MagConv2ClpActIdle;

				tyP0939MagConv4.tyFB.tyBtnRemoteUnclamp.bValue	:= FALSE;

			ELSIF p_eMagConv2Clp4Status = Error THEN

				tyP0939MagConv4.tyFB.tyBtnRemoteUnclamp.bValue	:= FALSE;

			END_IF

		ELSIF tyP0939MagConv4.tyFB.tyBtnRemoteClamp.bValue = TRUE THEN
			eMagConv2Clp4Act	:= MagConv2ClpActRmtClprClamp;

			IF p_eMagConv2Clp4Stat = MagConv2ClpActRmtClprClamp AND p_eMagConv2Clp4Status = Done THEN

				eMagConv2Clp4Act	:= MagConv2ClpActIdle;

				tyP0939MagConv4.tyFB.tyBtnRemoteClamp.bValue := FALSE;

			ELSIF p_eMagConv2Clp4Status = Error THEN
				tyP0939MagConv4.tyFB.tyBtnRemoteClamp.bValue := FALSE;

			END_IF

		END_IF

		//Selection Clamper
		IF tyP0939MagConv4.tyFB.tyBtnSelUnclamp.bValue = TRUE THEN

			eMagConvSelClp4Act	:= PneuActExt;

			IF p_eSelClamp4Stat = PneuActExt AND p_eSelClamp4Status = Done THEN

				eMagConvSelClp4Act	:= PneuActIdle;

				tyP0939MagConv4.tyFB.tyBtnSelUnclamp.bValue	:= FALSE;

			ELSIF p_eSelClamp4Status = Error THEN
				eMagConvSelClp4Act	:= PneuActIdle;
				tyP0939MagConv4.tyFB.tyBtnSelUnclamp.bValue	:= FALSE;

			END_IF

		ELSIF tyP0939MagConv4.tyFB.tyBtnSelClamp.bValue = TRUE THEN
			eMagConvSelClp4Act	:= PneuActRet;

			IF p_eSelClamp4Stat = PneuActRet AND p_eSelClamp4Status = Done THEN

				eMagConvSelClp4Act	:= PneuActIdle;

				tyP0939MagConv4.tyFB.tyBtnSelClamp.bValue	:= FALSE;

			ELSIF p_eSelClamp4Status = Error THEN
				eMagConvSelClp4Act	:= PneuActIdle;
				tyP0939MagConv4.tyFB.tyBtnSelClamp.bValue	:= FALSE;

			END_IF

		END_IF

		//Update Status
		tyP0939MagConv4.tyDC.tyBtnFixedUnclamp.bValue	:= NOT p_bMagConv2Clp4ClprFixClampCtrl;
		tyP0939MagConv4.tyDC.tyBtnFixedClamp.bValue		:= p_bMagConv2Clp4ClprFixClampCtrl;
		tyP0939MagConv4.tyDC.tyBtnRemoteUnclamp.bValue	:= NOT p_bMagConv2Clp4ClprRmtClampCtrl;
		tyP0939MagConv4.tyDC.tyBtnRemoteClamp.bValue	:= p_bMagConv2Clp4ClprRmtClampCtrl;

		tyP0939MagConv4.tyDC.tyBtnSelUnclamp.bRtCompl	:= FALSE;
		tyP0939MagConv4.tyDC.tyBtnSelClamp.bRtCompl		:= FALSE;
		tyP0939MagConv4.tyDC.tyBtnSelUnclamp.bValue	:= p_bSelClamp4RetCtrl;
		tyP0939MagConv4.tyDC.tyBtnSelClamp.bValue	:= p_bSelClamp4ExtCtrl;
	END_IF

	//Mask
	IF p_tyUsrMgmtCurrAccessRgt.bManualFBOnly THEN

		fUIInRtStatOff(ADR(tyP0939MagConv4.tyCom.tyBtnSwitch.uiMaskRtStat));

	ELSE

		IF p_eMagConv2Clp4Status = Error THEN

			fUIInRtStatOff(ADR(tyP0939MagConv4.tyFB.tyBtnEnt.uiMaskRtStat));
			fUIInRtStatOff(ADR(tyP0939MagConv4.tyFB.tyBtnExit.uiMaskRtStat));
			fUIInRtStatOff(ADR(tyP0939MagConv4.tyFB.tyBtnFixedClamp.uiMaskRtStat));
			fUIInRtStatOff(ADR(tyP0939MagConv4.tyFB.tyBtnFixedUnclamp.uiMaskRtStat));
			fUIInRtStatOff(ADR(tyP0939MagConv4.tyFB.tyBtnRemoteClamp.uiMaskRtStat));
			fUIInRtStatOff(ADR(tyP0939MagConv4.tyFB.tyBtnRemoteUnclamp.uiMaskRtStat));
			fUIInRtStatOff(ADR(tyP0939MagConv4.tyFB.tyBtnSelClamp.uiMaskRtStat));
			fUIInRtStatOff(ADR(tyP0939MagConv4.tyFB.tyBtnSelUnclamp.uiMaskRtStat));
			fUIInRtStatHide(ADR(tyP0939MagConv4.tyCom.tyBtnSwitch.uiMaskRtStat));

		ELSIF tyP0939MagConv4.tyFB.tyBtnEnt.bRtCompl = TRUE THEN

			fUIInRtStatHide(ADR(tyP0939MagConv4.tyFB.tyBtnEnt.uiMaskRtStat));
			fUIInRtStatOff(ADR(tyP0939MagConv4.tyFB.tyBtnExit.uiMaskRtStat));
			fUIInRtStatOff(ADR(tyP0939MagConv4.tyFB.tyBtnFixedClamp.uiMaskRtStat));
			fUIInRtStatOff(ADR(tyP0939MagConv4.tyFB.tyBtnFixedUnclamp.uiMaskRtStat));
			fUIInRtStatOff(ADR(tyP0939MagConv4.tyFB.tyBtnRemoteClamp.uiMaskRtStat));
			fUIInRtStatOff(ADR(tyP0939MagConv4.tyFB.tyBtnRemoteUnclamp.uiMaskRtStat));
			fUIInRtStatOff(ADR(tyP0939MagConv4.tyFB.tyBtnSelClamp.uiMaskRtStat));
			fUIInRtStatOff(ADR(tyP0939MagConv4.tyFB.tyBtnSelUnclamp.uiMaskRtStat));
			fUIInRtStatOff(ADR(tyP0939MagConv4.tyCom.tyBtnSwitch.uiMaskRtStat));

		ELSIF tyP0939MagConv4.tyFB.tyBtnExit.bRtCompl = TRUE THEN

			fUIInRtStatOff(ADR(tyP0939MagConv4.tyFB.tyBtnEnt.uiMaskRtStat));
			fUIInRtStatHide(ADR(tyP0939MagConv4.tyFB.tyBtnExit.uiMaskRtStat));
			fUIInRtStatOff(ADR(tyP0939MagConv4.tyFB.tyBtnFixedClamp.uiMaskRtStat));
			fUIInRtStatOff(ADR(tyP0939MagConv4.tyFB.tyBtnFixedUnclamp.uiMaskRtStat));
			fUIInRtStatOff(ADR(tyP0939MagConv4.tyFB.tyBtnRemoteClamp.uiMaskRtStat));
			fUIInRtStatOff(ADR(tyP0939MagConv4.tyFB.tyBtnRemoteUnclamp.uiMaskRtStat));
			fUIInRtStatOff(ADR(tyP0939MagConv4.tyFB.tyBtnSelClamp.uiMaskRtStat));
			fUIInRtStatOff(ADR(tyP0939MagConv4.tyFB.tyBtnSelUnclamp.uiMaskRtStat));
			fUIInRtStatOff(ADR(tyP0939MagConv4.tyCom.tyBtnSwitch.uiMaskRtStat));

		ELSIF tyP0939MagConv4.tyFB.tyBtnFixedClamp.bValue = TRUE OR tyP0939MagConv4.tyFB.tyBtnRemoteClamp.bValue = TRUE
			OR tyP0939MagConv4.tyFB.tyBtnFixedUnclamp.bValue = TRUE OR tyP0939MagConv4.tyFB.tyBtnRemoteUnclamp.bValue = TRUE
			OR tyP0939MagConv4.tyFB.tyBtnSelClamp.bValue = TRUE OR tyP0939MagConv4.tyFB.tyBtnSelUnclamp.bValue = TRUE
			THEN

			fUIInRtStatOff(ADR(tyP0939MagConv4.tyFB.tyBtnEnt.uiMaskRtStat));
			fUIInRtStatOff(ADR(tyP0939MagConv4.tyFB.tyBtnExit.uiMaskRtStat));
			fUIInRtStatHide(ADR(tyP0939MagConv4.tyFB.tyBtnFixedClamp.uiMaskRtStat));
			fUIInRtStatHide(ADR(tyP0939MagConv4.tyFB.tyBtnFixedUnclamp.uiMaskRtStat));
			fUIInRtStatHide(ADR(tyP0939MagConv4.tyFB.tyBtnRemoteClamp.uiMaskRtStat));
			fUIInRtStatHide(ADR(tyP0939MagConv4.tyFB.tyBtnRemoteUnclamp.uiMaskRtStat));
			fUIInRtStatHide(ADR(tyP0939MagConv4.tyFB.tyBtnSelClamp.uiMaskRtStat));
			fUIInRtStatHide(ADR(tyP0939MagConv4.tyFB.tyBtnSelUnclamp.uiMaskRtStat));
			fUIInRtStatOff(ADR(tyP0939MagConv4.tyCom.tyBtnSwitch.uiMaskRtStat));

		ELSE

			fUIInRtStatHide(ADR(tyP0939MagConv4.tyFB.tyBtnEnt.uiMaskRtStat));
			fUIInRtStatHide(ADR(tyP0939MagConv4.tyFB.tyBtnExit.uiMaskRtStat));
			fUIInRtStatHide(ADR(tyP0939MagConv4.tyFB.tyBtnFixedClamp.uiMaskRtStat));
			fUIInRtStatHide(ADR(tyP0939MagConv4.tyFB.tyBtnFixedUnclamp.uiMaskRtStat));
			fUIInRtStatHide(ADR(tyP0939MagConv4.tyFB.tyBtnRemoteClamp.uiMaskRtStat));
			fUIInRtStatHide(ADR(tyP0939MagConv4.tyFB.tyBtnRemoteUnclamp.uiMaskRtStat));
			fUIInRtStatHide(ADR(tyP0939MagConv4.tyFB.tyBtnSelClamp.uiMaskRtStat));
			fUIInRtStatHide(ADR(tyP0939MagConv4.tyFB.tyBtnSelUnclamp.uiMaskRtStat));
			fUIInRtStatHide(ADR(tyP0939MagConv4.tyCom.tyBtnSwitch.uiMaskRtStat));

		END_IF
	END_IF

	IF p_tyDI.bMagConvCAB717MagSen4 THEN
		fUIInRtStatOff(ADR(tyP0939MagConv4.tyFB.tyBtnSelClamp.uiMaskRtStat));
	END_IF

END_ACTION
```

#### Act_OptP0939MagConv4FBStat.st
```iecst
ACTION Act_OptP0939MagConv4FBStat:

	IF tyP0939MagConv4.tyFB.tyBtnFixedClamp.bValue = TRUE OR tyP0939MagConv4.tyFB.tyBtnRemoteClamp.bValue = TRUE
		OR tyP0939MagConv4.tyFB.tyBtnFixedUnclamp.bValue = TRUE OR tyP0939MagConv4.tyFB.tyBtnRemoteUnclamp.bValue = TRUE
		THEN
		tyP0939MagConv4.tyFB.tyStringStat.sValue	:= p_sMagConv2Clp4StatTxt;
	ELSIF tyP0939MagConv4.tyFB.tyBtnSelUnclamp.bValue = TRUE OR tyP0939MagConv4.tyFB.tyBtnSelClamp.bValue = TRUE
		THEN
		tyP0939MagConv4.tyFB.tyStringStat.sValue	:= p_sSelClamp4StatTxt;
	END_IF
END_ACTION
```

#### Act_OptP0939MagConv4DC.st
```iecst
ACTION Act_OptP0939MagConv4DC:

	//Magazine Conveyor
	IF tyP0939MagConv4.tyDC.tyBtnStop.bRtCompl = TRUE THEN
		eMagConv2Clp4Act	:= MagConv2ClpActStop;

		IF p_eMagConv2Clp4Stat = MagConv2ClpActStop AND p_eMagConv2Clp4Status = Done THEN
			eMagConv2Clp4Act	:= MagConv2ClpActIdle;

			tyP0939MagConv4.tyDC.tyBtnStop.bRtCompl		:= FALSE;
			tyP0939MagConv4.tyDC.tyBtnStop.bValue		:= TRUE;
			tyP0939MagConv4.tyDC.tyBtnStop.bRtLk		:= TRUE;

			tyP0939MagConv4.tyDC.tyBtnMagIn.bRtCompl	:= FALSE;
			tyP0939MagConv4.tyDC.tyBtnMagIn.bValue		:= FALSE;
			tyP0939MagConv4.tyDC.tyBtnMagIn.bRtLk		:= FALSE;

			tyP0939MagConv4.tyDC.tyBtnMagOut.bRtCompl	:= FALSE;
			tyP0939MagConv4.tyDC.tyBtnMagOut.bValue		:= FALSE;
			tyP0939MagConv4.tyDC.tyBtnMagOut.bRtLk		:= FALSE;
		END_IF

	ELSIF tyP0939MagConv4.tyDC.tyBtnMagIn.bRtCompl = TRUE THEN
		tyP0939MagConv4.tyDC.tyBtnMagIn.bValue	:= TRUE;
		tyP0939MagConv4.tyDC.tyBtnMagIn.bRtLk	:= TRUE;

		tyP0939MagConv4.tyDC.tyBtnStop.bValue	:= FALSE;
		tyP0939MagConv4.tyDC.tyBtnStop.bRtLk	:= FALSE;

		IF p_tyNtParamCurr.eProjMagConvDir = ConvDirLToR OR p_tyNtParamCurr.eProjMagConvDir = ConvDirLToL THEN

			eMagConv2Clp4Act	:= MagConv2ClpActSetMtrSigOnOrLToR;

			IF p_eMagConv2Clp4Stat = MagConv2ClpActSetMtrSigOnOrLToR AND p_eMagConv2Clp4Status = Done THEN
				eMagConv2Clp4Act	:= MagConv2ClpActIdle;

				tyP0939MagConv4.tyDC.tyBtnMagIn.bRtCompl	:= FALSE;
			END_IF

		ELSE

			eMagConv2Clp4Act	:= MagConv2ClpActSetMtrDirOrRToL;

			IF p_eMagConv2Clp4Stat = MagConv2ClpActSetMtrDirOrRToL AND p_eMagConv2Clp4Status = Done THEN
				eMagConv2Clp4Act	:= MagConv2ClpActIdle;

				tyP0939MagConv4.tyDC.tyBtnMagIn.bRtCompl	:= FALSE;
			END_IF

		END_IF

	ELSIF tyP0939MagConv4.tyDC.tyBtnMagOut.bRtCompl = TRUE THEN
		tyP0939MagConv4.tyDC.tyBtnMagOut.bValue	:= TRUE;
		tyP0939MagConv4.tyDC.tyBtnMagOut.bRtLk	:= TRUE;

		tyP0939MagConv4.tyDC.tyBtnStop.bValue	:= FALSE;
		tyP0939MagConv4.tyDC.tyBtnStop.bRtLk	:= FALSE;

		IF p_tyNtParamCurr.eProjMagConvDir = ConvDirLToR OR p_tyNtParamCurr.eProjMagConvDir = ConvDirRToR THEN

			eMagConv2Clp4Act	:= MagConv2ClpActSetMtrSigOnOrLToR;

			IF p_eMagConv2Clp4Stat = MagConv2ClpActSetMtrSigOnOrLToR AND p_eMagConv2Clp4Status = Done THEN
				eMagConv2Clp4Act	:= MagConv2ClpActIdle;

				tyP0939MagConv4.tyDC.tyBtnMagOut.bRtCompl	:= FALSE;
			END_IF

		ELSE

			eMagConv2Clp4Act	:= MagConv2ClpActSetMtrDirOrRToL;

			IF p_eMagConv2Clp4Stat = MagConv2ClpActSetMtrDirOrRToL AND p_eMagConv2Clp4Status = Done THEN
				eMagConv2Clp4Act	:= MagConv2ClpActIdle;

				tyP0939MagConv4.tyDC.tyBtnMagOut.bRtCompl	:= FALSE;
			END_IF

		END_IF

	END_IF

	//Magazine Clamper
	IF tyP0939MagConv4.tyCom.tyBtnSwitch.bValue = TRUE THEN
		IF p_bSelClamp4TwoCtrlOut = FALSE THEN
			IF tyP0939MagConv4.tyDC.tyBtnSelUnclamp.bRtCompl = TRUE THEN
				tyP0939MagConv4.tyDC.tyBtnSelUnclamp.bValue := TRUE;
				tyP0939MagConv4.tyDC.tyBtnSelClamp.bValue := FALSE;

				eMagConvSelClp4Act	:= PneuActSetExt;

				IF p_eSelClamp4Stat = PneuActSetExt AND p_eSelClamp4Status = Done THEN
					eMagConvSelClp4Act	:= PneuActIdle;

					tyP0939MagConv4.tyDC.tyBtnSelUnclamp.bRtCompl	:= FALSE;
				END_IF

			ELSIF tyP0939MagConv4.tyDC.tyBtnSelClamp.bRtCompl = TRUE THEN
				tyP0939MagConv4.tyDC.tyBtnSelClamp.bValue := TRUE;
				tyP0939MagConv4.tyDC.tyBtnSelUnclamp.bValue := FALSE;

				eMagConvSelClp4Act	:= PneuActSetRet;

				IF p_eSelClamp4Stat = PneuActSetRet AND p_eSelClamp4Status = Done THEN
					eMagConvSelClp4Act	:= PneuActIdle;

					tyP0939MagConv4.tyDC.tyBtnSelClamp.bRtCompl	:= FALSE;
				END_IF
			END_IF

		ELSE
			IF (tyP0939MagConv4.tyDC.tyBtnSelUnclamp.bRtCompl = TRUE) OR (tyP0939MagConv4.tyDC.tyBtnSelClamp.bRtCompl = TRUE) THEN
				IF (tyP0939MagConv4.tyDC.tyBtnSelUnclamp.bValue = TRUE) AND (tyP0939MagConv4.tyDC.tyBtnSelClamp.bValue = TRUE) THEN
					eMagConvSelClp4Act	:= PneuActSetAll;

					IF p_eSelClamp4Stat = PneuActSetAll AND p_eSelClamp4Status = Done THEN
						eMagConvSelClp4Act	:= PneuActIdle;

						tyP0939MagConv4.tyDC.tyBtnSelUnclamp.bRtCompl		:= FALSE;
						tyP0939MagConv4.tyDC.tyBtnSelClamp.bRtCompl			:= FALSE;
					END_IF

				ELSIF (tyP0939MagConv4.tyDC.tyBtnSelUnclamp.bValue = TRUE) AND (tyP0939MagConv4.tyDC.tyBtnSelClamp.bValue = FALSE) THEN
					eMagConvSelClp4Act	:= PneuActSetExt;

					IF p_eSelClamp4Stat = PneuActSetExt AND p_eSelClamp4Status = Done THEN
						eMagConvSelClp4Act	:= PneuActIdle;

						tyP0939MagConv4.tyDC.tyBtnSelUnclamp.bRtCompl		:= FALSE;
						tyP0939MagConv4.tyDC.tyBtnSelClamp.bRtCompl			:= FALSE;
					END_IF

				ELSIF (tyP0939MagConv4.tyDC.tyBtnSelUnclamp.bValue = FALSE) AND (tyP0939MagConv4.tyDC.tyBtnSelClamp.bValue = TRUE) THEN
					eMagConvSelClp4Act	:= PneuActSetRet;

					IF p_eSelClamp4Stat = PneuActSetRet AND p_eSelClamp4Status = Done THEN
						eMagConvSelClp4Act	:= PneuActIdle;

						tyP0939MagConv4.tyDC.tyBtnSelUnclamp.bRtCompl		:= FALSE;
						tyP0939MagConv4.tyDC.tyBtnSelClamp.bRtCompl			:= FALSE;
					END_IF

				ELSE
					eMagConvSelClp4Act	:= PneuActRstAll;

					IF p_eSelClamp4Stat = PneuActRstAll AND p_eSelClamp4Status = Done THEN
						eMagConvSelClp4Act	:= PneuActIdle;

						tyP0939MagConv4.tyDC.tyBtnSelUnclamp.bRtCompl		:= FALSE;
						tyP0939MagConv4.tyDC.tyBtnSelClamp.bRtCompl			:= FALSE;
					END_IF

				END_IF
			END_IF
		END_IF
		IF p_bMagConv2Clp1ClprTwoOutputCtrl = FALSE THEN

			//Fixed
			IF tyP0939MagConv4.tyDC.tyBtnFixedClamp.bRtCompl = TRUE THEN
				tyP0939MagConv4.tyDC.tyBtnFixedClamp.bValue		:= TRUE;
				tyP0939MagConv4.tyDC.tyBtnFixedUnclamp.bValue	:= FALSE;

				eMagConv2Clp4Act	:= MagConv2ClpActFixClprSetClamp;

				IF p_eMagConv2Clp4Stat = MagConv2ClpActFixClprSetClamp AND p_eMagConv2Clp4Status = Done THEN
					eMagConv2Clp4Act	:= MagConv2ClpActIdle;

					tyP0939MagConv4.tyDC.tyBtnFixedClamp.bRtCompl	:= FALSE;
				END_IF

			ELSIF tyP0939MagConv4.tyDC.tyBtnFixedUnclamp.bRtCompl = TRUE THEN
				tyP0939MagConv4.tyDC.tyBtnFixedUnclamp.bValue	:= TRUE;
				tyP0939MagConv4.tyDC.tyBtnFixedClamp.bValue		:= FALSE;

				eMagConv2Clp4Act	:= MagConv2ClpActFixClprSetUnclamp;

				IF p_eMagConv2Clp4Stat = MagConv2ClpActFixClprSetUnclamp AND p_eMagConv2Clp4Status = Done THEN
					eMagConv2Clp4Act	:= MagConv2ClpActIdle;

					tyP0939MagConv4.tyDC.tyBtnFixedUnclamp.bRtCompl	:= FALSE;
				END_IF

			END_IF

			//Remote
			IF tyP0939MagConv4.tyDC.tyBtnRemoteClamp.bRtCompl = TRUE THEN
				tyP0939MagConv4.tyDC.tyBtnRemoteClamp.bValue		:= TRUE;
				tyP0939MagConv4.tyDC.tyBtnRemoteUnclamp.bValue		:= FALSE;

				eMagConv2Clp4Act	:= MagConv2ClpActRmtClprSetClamp;

				IF p_eMagConv2Clp4Stat = MagConv2ClpActRmtClprSetClamp AND p_eMagConv2Clp4Status = Done THEN
					eMagConv2Clp4Act	:= MagConv2ClpActIdle;

					tyP0939MagConv4.tyDC.tyBtnRemoteClamp.bRtCompl	:= FALSE;
				END_IF

			ELSIF tyP0939MagConv4.tyDC.tyBtnRemoteUnclamp.bRtCompl = TRUE THEN
				tyP0939MagConv4.tyDC.tyBtnRemoteUnclamp.bValue	:= TRUE;
				tyP0939MagConv4.tyDC.tyBtnRemoteClamp.bValue	:= FALSE;

				eMagConv2Clp4Act	:= MagConv2ClpActRmtClprSetUnclamp;

				IF p_eMagConv2Clp4Stat = MagConv2ClpActRmtClprSetUnclamp AND p_eMagConv2Clp4Status = Done THEN
					eMagConv2Clp4Act	:= MagConv2ClpActIdle;

					tyP0939MagConv4.tyDC.tyBtnRemoteUnclamp.bRtCompl	:= FALSE;
				END_IF

			END_IF

		ELSE

			//Fixed
			IF (tyP0939MagConv4.tyDC.tyBtnFixedClamp.bRtCompl = TRUE) OR (tyP0939MagConv4.tyDC.tyBtnFixedUnclamp.bRtCompl = TRUE) THEN

				IF (tyP0939MagConv4.tyDC.tyBtnFixedClamp.bValue = TRUE) AND (tyP0939MagConv4.tyDC.tyBtnFixedUnclamp.bValue = TRUE) THEN

					eMagConv2Clp4Act	:= MagConv2ClpActFixClprSetAll;

					IF p_eMagConv2Clp4Stat = MagConv2ClpActFixClprSetAll AND p_eMagConv2Clp4Status = Done THEN

						eMagConv2Clp4Act	:= MagConv2ClpActIdle;

						tyP0939MagConv4.tyDC.tyBtnFixedClamp.bRtCompl	:= FALSE;
						tyP0939MagConv4.tyDC.tyBtnFixedUnclamp.bRtCompl	:= FALSE;
					END_IF

				ELSIF (tyP0939MagConv4.tyDC.tyBtnFixedClamp.bValue = TRUE) AND (tyP0939MagConv4.tyDC.tyBtnFixedUnclamp.bValue = FALSE) THEN
					eMagConv2Clp4Act	:= MagConv2ClpActFixClprSetClamp;

					IF p_eMagConv2Clp4Stat = MagConv2ClpActFixClprSetClamp AND p_eMagConv2Clp4Status = Done THEN

						eMagConv2Clp4Act	:= MagConv2ClpActIdle;

						tyP0939MagConv4.tyDC.tyBtnFixedClamp.bRtCompl	:= FALSE;
						tyP0939MagConv4.tyDC.tyBtnFixedUnclamp.bRtCompl	:= FALSE;
					END_IF

				ELSIF (tyP0939MagConv4.tyDC.tyBtnFixedClamp.bValue = FALSE) AND (tyP0939MagConv4.tyDC.tyBtnFixedUnclamp.bValue = TRUE) THEN
					eMagConv2Clp4Act	:= MagConv2ClpActFixClprSetUnclamp;

					IF p_eMagConv2Clp4Stat = MagConv2ClpActFixClprSetUnclamp AND p_eMagConv2Clp4Status = Done THEN

						eMagConv2Clp4Act	:= MagConv2ClpActIdle;

						tyP0939MagConv4.tyDC.tyBtnFixedClamp.bRtCompl	:= FALSE;
						tyP0939MagConv4.tyDC.tyBtnFixedUnclamp.bRtCompl	:= FALSE;
					END_IF

				ELSE
					eMagConv2Clp4Act	:= MagConv2ClpActFixClprRstAll;

					IF p_eMagConv2Clp4Stat = MagConv2ClpActFixClprRstAll AND p_eMagConv2Clp4Status = Done THEN

						eMagConv2Clp4Act	:= MagConv2ClpActIdle;

						tyP0939MagConv4.tyDC.tyBtnFixedClamp.bRtCompl	:= FALSE;
						tyP0939MagConv4.tyDC.tyBtnFixedUnclamp.bRtCompl	:= FALSE;
					END_IF

				END_IF

				//Remote
				IF (tyP0939MagConv4.tyDC.tyBtnRemoteClamp.bRtCompl = TRUE) OR (tyP0939MagConv4.tyDC.tyBtnRemoteUnclamp.bRtCompl = TRUE) THEN

					IF (tyP0939MagConv4.tyDC.tyBtnRemoteClamp.bValue = TRUE) AND (tyP0939MagConv4.tyDC.tyBtnRemoteUnclamp.bValue = TRUE) THEN

						eMagConv2Clp4Act	:= MagConv2ClpActRmtClprSetAll;

						IF p_eMagConv2Clp4Stat = MagConv2ClpActRmtClprSetAll AND p_eMagConv2Clp4Status = Done THEN

							eMagConv2Clp4Act	:= MagConv2ClpActIdle;

							tyP0939MagConv4.tyDC.tyBtnRemoteClamp.bRtCompl		:= FALSE;
							tyP0939MagConv4.tyDC.tyBtnRemoteUnclamp.bRtCompl	:= FALSE;
						END_IF

					ELSIF (tyP0939MagConv4.tyDC.tyBtnRemoteClamp.bValue = TRUE) AND (tyP0939MagConv4.tyDC.tyBtnRemoteUnclamp.bValue = FALSE) THEN
						eMagConv2Clp4Act	:= MagConv2ClpActRmtClprSetClamp;

						IF p_eMagConv2Clp4Stat = MagConv2ClpActRmtClprSetClamp AND p_eMagConv2Clp4Status = Done THEN

							eMagConv2Clp4Act	:= MagConv2ClpActIdle;

							tyP0939MagConv4.tyDC.tyBtnRemoteClamp.bRtCompl	:= FALSE;
							tyP0939MagConv4.tyDC.tyBtnRemoteUnclamp.bRtCompl	:= FALSE;
						END_IF

					ELSIF (tyP0939MagConv4.tyDC.tyBtnRemoteClamp.bValue = FALSE) AND (tyP0939MagConv4.tyDC.tyBtnRemoteUnclamp.bValue = TRUE) THEN
						eMagConv2Clp4Act	:= MagConv2ClpActRmtClprSetUnclamp;

						IF p_eMagConv2Clp4Stat = MagConv2ClpActRmtClprSetUnclamp AND p_eMagConv2Clp4Status = Done THEN

							eMagConv2Clp4Act	:= MagConv2ClpActIdle;

							tyP0939MagConv4.tyDC.tyBtnRemoteClamp.bRtCompl	:= FALSE;
							tyP0939MagConv4.tyDC.tyBtnRemoteUnclamp.bRtCompl	:= FALSE;
						END_IF

					ELSE
						eMagConv2Clp4Act	:= MagConv2ClpActRmtClprRstAll;

						IF p_eMagConv2Clp4Stat = MagConv2ClpActRmtClprRstAll AND p_eMagConv2Clp4Status = Done THEN

							eMagConv2Clp4Act	:= MagConv2ClpActIdle;

							tyP0939MagConv4.tyDC.tyBtnRemoteClamp.bRtCompl	:= FALSE;
							tyP0939MagConv4.tyDC.tyBtnRemoteUnclamp.bRtCompl	:= FALSE;
						END_IF

					END_IF
				END_IF

			END_IF

		END_IF

		//Fixed
		tyP0939MagConv4.tyFB.tyBtnFixedClamp.bRtCompl		:= FALSE;
		tyP0939MagConv4.tyFB.tyBtnFixedClamp.bValue			:= FALSE;
		tyP0939MagConv4.tyFB.tyBtnFixedUnclamp.bRtCompl		:= FALSE;
		tyP0939MagConv4.tyFB.tyBtnFixedUnclamp.bValue		:= FALSE;

		//Remote
		tyP0939MagConv4.tyFB.tyBtnRemoteClamp.bRtCompl		:= FALSE;
		tyP0939MagConv4.tyFB.tyBtnRemoteClamp.bValue		:= FALSE;
		tyP0939MagConv4.tyFB.tyBtnRemoteUnclamp.bRtCompl	:= FALSE;
		tyP0939MagConv4.tyFB.tyBtnRemoteUnclamp.bValue		:= FALSE;

	END_IF

	//Mask
	IF p_eMagConv2Clp4Status = Error THEN

		fUIInRtStatOff(ADR(tyP0939MagConv4.tyDC.tyBtnMagIn.uiMaskRtStat));
		fUIInRtStatOff(ADR(tyP0939MagConv4.tyDC.tyBtnMagOut.uiMaskRtStat));
		fUIInRtStatOff(ADR(tyP0939MagConv4.tyDC.tyBtnFixedClamp.uiMaskRtStat));
		fUIInRtStatOff(ADR(tyP0939MagConv4.tyDC.tyBtnFixedUnclamp.uiMaskRtStat));
		fUIInRtStatOff(ADR(tyP0939MagConv4.tyDC.tyBtnRemoteClamp.uiMaskRtStat));
		fUIInRtStatOff(ADR(tyP0939MagConv4.tyDC.tyBtnRemoteUnclamp.uiMaskRtStat));

	ELSIF tyP0939MagConv4.tyDC.tyBtnMagIn.bValue = TRUE THEN

		fUIInRtStatHide(ADR(tyP0939MagConv4.tyDC.tyBtnMagIn.uiMaskRtStat));
		fUIInRtStatOff(ADR(tyP0939MagConv4.tyDC.tyBtnMagOut.uiMaskRtStat));
		fUIInRtStatOff(ADR(tyP0939MagConv4.tyDC.tyBtnFixedClamp.uiMaskRtStat));
		fUIInRtStatOff(ADR(tyP0939MagConv4.tyDC.tyBtnFixedUnclamp.uiMaskRtStat));
		fUIInRtStatOff(ADR(tyP0939MagConv4.tyDC.tyBtnRemoteClamp.uiMaskRtStat));
		fUIInRtStatOff(ADR(tyP0939MagConv4.tyDC.tyBtnRemoteUnclamp.uiMaskRtStat));

	ELSIF tyP0939MagConv4.tyDC.tyBtnMagOut.bValue = TRUE THEN

		fUIInRtStatOff(ADR(tyP0939MagConv4.tyDC.tyBtnMagIn.uiMaskRtStat));
		fUIInRtStatHide(ADR(tyP0939MagConv4.tyDC.tyBtnMagOut.uiMaskRtStat));
		fUIInRtStatOff(ADR(tyP0939MagConv4.tyDC.tyBtnFixedClamp.uiMaskRtStat));
		fUIInRtStatOff(ADR(tyP0939MagConv4.tyDC.tyBtnFixedUnclamp.uiMaskRtStat));
		fUIInRtStatOff(ADR(tyP0939MagConv4.tyDC.tyBtnRemoteClamp.uiMaskRtStat));
		fUIInRtStatOff(ADR(tyP0939MagConv4.tyDC.tyBtnRemoteUnclamp.uiMaskRtStat));

	ELSE

		fUIInRtStatHide(ADR(tyP0939MagConv4.tyDC.tyBtnMagIn.uiMaskRtStat));
		fUIInRtStatHide(ADR(tyP0939MagConv4.tyDC.tyBtnMagOut.uiMaskRtStat));
		fUIInRtStatHide(ADR(tyP0939MagConv4.tyDC.tyBtnFixedClamp.uiMaskRtStat));
		fUIInRtStatHide(ADR(tyP0939MagConv4.tyDC.tyBtnFixedUnclamp.uiMaskRtStat));
		fUIInRtStatHide(ADR(tyP0939MagConv4.tyDC.tyBtnRemoteClamp.uiMaskRtStat));
		fUIInRtStatHide(ADR(tyP0939MagConv4.tyDC.tyBtnRemoteUnclamp.uiMaskRtStat));

	END_IF

END_ACTION
```

#### Act_OptP0939RstMnl.st
```iecst
ACTION Act_OptP0939RstMnl:

	IF EDGEPOS((bManualMod = FALSE) OR (p_eMagConv2Clp4Status = Error)) THEN

		eMagConv2Clp4Act	:= MagConv2ClpActIdle;
		eMagConvSelClp4Act	:= PneuActIdle;
		//Magazine Conveyor
		//FB
		tyP0939MagConv4.tyFB.tyBtnEnt.bRtCompl				:= FALSE;
		tyP0939MagConv4.tyFB.tyBtnExit.bRtCompl				:= FALSE;
		tyP0939MagConv4.tyFB.tyBtnStop.bRtCompl				:= FALSE;

		tyP0939MagConv4.tyFB.tyBtnEnt.bValue				:= FALSE;
		tyP0939MagConv4.tyFB.tyBtnExit.bValue				:= FALSE;
		tyP0939MagConv4.tyFB.tyBtnStop.bValue				:= TRUE;

		tyP0939MagConv4.tyFB.tyBtnEnt.bRtLk					:= FALSE;
		tyP0939MagConv4.tyFB.tyBtnExit.bRtLk				:= FALSE;
		tyP0939MagConv4.tyFB.tyBtnStop.bRtLk				:= TRUE;

		tyP0939MagConv4.tyFB.tyBtnEnt.uiMaskRtStat.0		:= TRUE;
		tyP0939MagConv4.tyFB.tyBtnExit.uiMaskRtStat.0		:= TRUE;
		tyP0939MagConv4.tyCom.tyBtnSwitch.uiMaskRtStat.0	:= TRUE;

		//Direct
		tyP0939MagConv4.tyDC.tyBtnMagIn.bRtCompl			:= FALSE;
		tyP0939MagConv4.tyDC.tyBtnMagOut.bRtCompl			:= FALSE;
		tyP0939MagConv4.tyDC.tyBtnStop.bRtCompl				:= FALSE;

		tyP0939MagConv4.tyDC.tyBtnMagIn.bValue				:= FALSE;
		tyP0939MagConv4.tyDC.tyBtnMagOut.bValue				:= FALSE;
		tyP0939MagConv4.tyDC.tyBtnStop.bValue				:= TRUE;

		tyP0939MagConv4.tyDC.tyBtnMagIn.bRtLk				:= FALSE;
		tyP0939MagConv4.tyDC.tyBtnMagOut.bRtLk				:= FALSE;
		tyP0939MagConv4.tyDC.tyBtnStop.bRtLk				:= TRUE;

		tyP0939MagConv4.tyDC.tyBtnMagIn.uiMaskRtStat.0		:= TRUE;
		tyP0939MagConv4.tyDC.tyBtnMagOut.uiMaskRtStat.0		:= TRUE;
		tyP0939MagConv4.tyCom.tyBtnSwitch.uiMaskRtStat.0	:= TRUE;

		//Magazine Clamper
		//FB
		//Fixed/Bottom
		tyP0939MagConv4.tyFB.tyBtnFixedClamp.bRtCompl			:= FALSE;
		tyP0939MagConv4.tyFB.tyBtnFixedUnclamp.bRtCompl			:= FALSE;

		tyP0939MagConv4.tyFB.tyBtnFixedClamp.bValue				:= FALSE;
		tyP0939MagConv4.tyFB.tyBtnFixedUnclamp.bValue			:= FALSE;

		//Remote/Top
		tyP0939MagConv4.tyFB.tyBtnRemoteClamp.bRtCompl			:= FALSE;
		tyP0939MagConv4.tyFB.tyBtnRemoteUnclamp.bRtCompl		:= FALSE;

		tyP0939MagConv4.tyFB.tyBtnRemoteClamp.bValue			:= FALSE;
		tyP0939MagConv4.tyFB.tyBtnRemoteUnclamp.bValue			:= FALSE;

		//Selection
		tyP0939MagConv4.tyFB.tyBtnSelClamp.bRtCompl			:= FALSE;
		tyP0939MagConv4.tyFB.tyBtnSelUnclamp.bRtCompl		:= FALSE;

		tyP0939MagConv4.tyFB.tyBtnSelClamp.bValue			:= FALSE;
		tyP0939MagConv4.tyFB.tyBtnSelUnclamp.bValue			:= FALSE;

		tyP0939MagConv4.tyFB.tyBtnFixedClamp.uiMaskRtStat.0		:= TRUE;
		tyP0939MagConv4.tyFB.tyBtnFixedUnclamp.uiMaskRtStat.0	:= TRUE;
		tyP0939MagConv4.tyFB.tyBtnRemoteClamp.uiMaskRtStat.0	:= TRUE;
		tyP0939MagConv4.tyFB.tyBtnRemoteUnclamp.uiMaskRtStat.0	:= TRUE;
		tyP0939MagConv4.tyFB.tyBtnSelClamp.uiMaskRtStat.0		:= TRUE;
		tyP0939MagConv4.tyFB.tyBtnSelUnclamp.uiMaskRtStat.0		:= TRUE;

		tyP0939MagConv4.tyCom.tyBtnSwitch.uiMaskRtStat.0		:= TRUE;

		//Direct
		//Fixed/Bottom
		tyP0939MagConv4.tyDC.tyBtnFixedClamp.bRtCompl			:= FALSE;
		tyP0939MagConv4.tyDC.tyBtnFixedUnclamp.bRtCompl			:= FALSE;

		tyP0939MagConv4.tyDC.tyBtnFixedClamp.bValue				:= FALSE;
		tyP0939MagConv4.tyDC.tyBtnFixedUnclamp.bValue			:= FALSE;

		//Remote/Top
		tyP0939MagConv4.tyDC.tyBtnRemoteClamp.bRtCompl			:= FALSE;
		tyP0939MagConv4.tyDC.tyBtnRemoteUnclamp.bRtCompl		:= FALSE;

		tyP0939MagConv4.tyDC.tyBtnRemoteClamp.bValue			:= FALSE;
		tyP0939MagConv4.tyDC.tyBtnRemoteUnclamp.bValue			:= FALSE;

		//Selection
		tyP0939MagConv4.tyDC.tyBtnSelClamp.bRtCompl				:= FALSE;
		tyP0939MagConv4.tyDC.tyBtnSelUnclamp.bRtCompl			:= FALSE;

		tyP0939MagConv4.tyDC.tyBtnSelClamp.bValue				:= FALSE;
		tyP0939MagConv4.tyDC.tyBtnSelUnclamp.bValue				:= FALSE;

		tyP0939MagConv4.tyDC.tyBtnFixedClamp.uiMaskRtStat.0		:= TRUE;
		tyP0939MagConv4.tyDC.tyBtnFixedUnclamp.uiMaskRtStat.0	:= TRUE;
		tyP0939MagConv4.tyDC.tyBtnRemoteClamp.uiMaskRtStat.0	:= TRUE;
		tyP0939MagConv4.tyDC.tyBtnRemoteUnclamp.uiMaskRtStat.0	:= TRUE;
		tyP0939MagConv4.tyDC.tyBtnSelClamp.uiMaskRtStat.0		:= TRUE;
		tyP0939MagConv4.tyDC.tyBtnSelUnclamp.uiMaskRtStat.0		:= TRUE;

		tyP0939MagConv4.tyCom.tyBtnSwitch.uiMaskRtStat.0		:= TRUE;

	END_IF

	IF EDGEPOS(bManualMod = FALSE) THEN
		tyP0939MagConv4.tyCom.tyBtnSwitch.bValue := FALSE;

		IF p_tyNtParamCurr.bMagAutoVerifyPrep = FALSE THEN
			fUIInRtStatHide(ADR(tyP0939MagConv4.tyDC.tyLyrWithoutSelClamp.uiRtStat));
			fUIInRtStatOff(ADR(tyP0939MagConv4.tyFB.tyLyrWithoutSelClamp.uiRtStat));
		ELSE

			fUIInRtStatHide(ADR(tyP0939MagConv4.tyDC.tyLyr.uiRtStat));
			fUIInRtStatOff(ADR(tyP0939MagConv4.tyFB.tyLyr.uiRtStat));
		END_IF

	END_IF

END_ACTION
```

#### Act_EntP0940Disp.st
```iecst
ACTION Act_EntP0940Disp:

	//Access Address
	p_tyC0005Main ACCESS ADR(tyCommon.tyMain);

	p_tyC0007Notif ACCESS ADR(tyCommon.tyNotif);

	p_tyC0008MsgBox ACCESS ADR(tyP0940CommCtrl.tyMsgBoxHide);

	p_tyC0009Info ACCESS ADR(tyCommon.tyInfo);

	p_tyP0940CommCtrlDSSMEMAA ACCESS ADR(tyP0940CommCtrl.tyDSSMEMAA);
	p_tyP0940CommCtrlDSSMEMAB ACCESS ADR(tyP0940CommCtrl.tyDSSMEMAB);
	p_tyP0940CommCtrlSOT ACCESS ADR(tyP0940CommCtrl.tySOT);

	CASE p_tyMcParamCurr.eAGVComProtocol OF
		McSetAGVCommOPCUA:
				tyP0940CommCtrl.tySOT.tyTxtAIVCommProtocol.usiValueIdx := 0;

		McSetAGVCommHardIO:
				tyP0940CommCtrl.tySOT.tyTxtAIVCommProtocol.usiValueIdx := 1;

		McSetAGVCommDisabled:
				tyP0940CommCtrl.tySOT.tyTxtAIVCommProtocol.usiValueIdx := 2;

	END_CASE

END_ACTION
```

#### Act_OptP0940ReadDI.st
```iecst
ACTION Act_OptP0940ReadDI:

	tyP0940CommCtrl.tyDSSMEMAA.tyBtnDSB.bValue	:= p_tyDI.bDSBA;
	tyP0940CommCtrl.tyDSSMEMAB.tyBtnDSB.bValue	:= p_tyDI.bDSBB;

	IF p_tyNtParamCurr.bProjSOTSensorPrep THEN
//		CASE p_tyMcParamCurr.eAGVComProtocol OF
//			McSetAGVCommHardIO:
				tyP0940CommCtrl.tySOT.tyBtnAIVRcv1.bValue		:= p_tyDI.bSOT1Receive;
				tyP0940CommCtrl.tySOT.tyBtnAIVErr1.bValue		:= p_tyDI.bSOT1AIVError;
				tyP0940CommCtrl.tySOT.tyBtnAIVRdy1.bValue		:= p_tyDI.bSOT1AIVReady;
				tyP0940CommCtrl.tySOT.tyBtnAIVAvail1.bValue		:= p_tyDI.bSOT1AIVAvailable;
				tyP0940CommCtrl.tySOT.tyBtnAIVSLarge1.bValue	:= p_tyDI.bSOT1AIVSizeLarge;

				tyP0940CommCtrl.tySOT.tyBtnAIVRcv2.bValue		:= p_tyDI.bSOT2Receive;
				tyP0940CommCtrl.tySOT.tyBtnAIVErr2.bValue		:= p_tyDI.bSOT2AIVError;
				tyP0940CommCtrl.tySOT.tyBtnAIVRdy2.bValue		:= p_tyDI.bSOT2AIVReady;
				tyP0940CommCtrl.tySOT.tyBtnAIVAvail2.bValue		:= p_tyDI.bSOT2AIVAvailable;
				tyP0940CommCtrl.tySOT.tyBtnAIVSLarge2.bValue	:= p_tyDI.bSOT2AIVSizeLarge;

				tyP0940CommCtrl.tySOT.tyBtnAIVRcv3.bValue		:= p_tyDI.bSOT3Receive;
				tyP0940CommCtrl.tySOT.tyBtnAIVErr3.bValue		:= p_tyDI.bSOT3AIVError;
				tyP0940CommCtrl.tySOT.tyBtnAIVRdy3.bValue		:= p_tyDI.bSOT3AIVReady;
				tyP0940CommCtrl.tySOT.tyBtnAIVAvail3.bValue		:= p_tyDI.bSOT3AIVAvailable;
				tyP0940CommCtrl.tySOT.tyBtnAIVSLarge3.bValue	:= p_tyDI.bSOT3AIVSizeLarge;

				tyP0940CommCtrl.tySOT.tyBtnAIVRcv4.bValue		:= p_tyDI.bSOT4Receive;
				tyP0940CommCtrl.tySOT.tyBtnAIVErr4.bValue		:= p_tyDI.bSOT4AIVError;
				tyP0940CommCtrl.tySOT.tyBtnAIVRdy4.bValue		:= p_tyDI.bSOT4AIVReady;
				tyP0940CommCtrl.tySOT.tyBtnAIVAvail4.bValue		:= p_tyDI.bSOT4AIVAvailable;
				tyP0940CommCtrl.tySOT.tyBtnAIVSLarge4.bValue	:= p_tyDI.bSOT4AIVSizeLarge;

				tyP0940CommCtrl.tySOT.tyBtnFleetMgrActive.bValue := p_tyDI.bFleetManagerReady OR p_tyTagFromMes.bActive;

//			McSetAGVCommOPCUA:
//
//				tyP0940CommCtrl.tySOT.tyBtnAIVErr1.bValue		:= p_tyTagFromMes.tyTagStatOfPlatforms[1].bError;
//				tyP0940CommCtrl.tySOT.tyBtnAIVRdy1.bValue		:= p_tyTagFromMes.tyTagStatOfPlatforms[1].bReady;
//				tyP0940CommCtrl.tySOT.tyBtnAIVAvail1.bValue		:= p_tyTagFromMes.tyTagStatOfPlatforms[1].bAvailable;
//				tyP0940CommCtrl.tySOT.tyBtnAIVSLarge1.bValue	:= p_tyTagFromMes.tyTagStatOfPlatforms[1].bSizeLarge;
//
//				tyP0940CommCtrl.tySOT.tyBtnAIVErr2.bValue		:= p_tyTagFromMes.tyTagStatOfPlatforms[2].bError;
//				tyP0940CommCtrl.tySOT.tyBtnAIVRdy2.bValue		:= p_tyTagFromMes.tyTagStatOfPlatforms[2].bReady;
//				tyP0940CommCtrl.tySOT.tyBtnAIVAvail2.bValue		:= p_tyTagFromMes.tyTagStatOfPlatforms[2].bAvailable;
//				tyP0940CommCtrl.tySOT.tyBtnAIVSLarge2.bValue	:= p_tyTagFromMes.tyTagStatOfPlatforms[2].bSizeLarge;
//
//				tyP0940CommCtrl.tySOT.tyBtnAIVErr3.bValue		:= p_tyTagFromMes.tyTagStatOfPlatforms[3].bError;
//				tyP0940CommCtrl.tySOT.tyBtnAIVRdy3.bValue		:= p_tyTagFromMes.tyTagStatOfPlatforms[3].bReady;
//				tyP0940CommCtrl.tySOT.tyBtnAIVAvail3.bValue		:= p_tyTagFromMes.tyTagStatOfPlatforms[3].bAvailable;
//				tyP0940CommCtrl.tySOT.tyBtnAIVSLarge3.bValue	:= p_tyTagFromMes.tyTagStatOfPlatforms[3].bSizeLarge;
//
//				tyP0940CommCtrl.tySOT.tyBtnAIVErr4.bValue		:= p_tyTagFromMes.tyTagStatOfPlatforms[4].bError;
//				tyP0940CommCtrl.tySOT.tyBtnAIVRdy4.bValue		:= p_tyTagFromMes.tyTagStatOfPlatforms[4].bReady;
//				tyP0940CommCtrl.tySOT.tyBtnAIVAvail4.bValue		:= p_tyTagFromMes.tyTagStatOfPlatforms[4].bAvailable;
//				tyP0940CommCtrl.tySOT.tyBtnAIVSLarge4.bValue	:= p_tyTagFromMes.tyTagStatOfPlatforms[4].bSizeLarge;
//
//				tyP0940CommCtrl.tySOT.tyBtnFleetMgrActive.bValue := p_tyTagFromMes.bActive;
//
//		END_CASE
	ELSIF p_tyMcParamCurr.eAGVComProtocol = McSetAGVCommHardIO AND p_tyNtParamCurr.bProjSOTSensorPrep = FALSE THEN
		tyP0940CommCtrl.tySOT.tyBtnAIVRcv1.bValue		:= p_tyDI.bSOT1Receive;
		tyP0940CommCtrl.tySOT.tyBtnAIVErr1.bValue		:= p_tyDI.bSOT1AIVError;
		tyP0940CommCtrl.tySOT.tyBtnAIVRdy1.bValue		:= p_tyDI.bSOT1AIVReady;
		tyP0940CommCtrl.tySOT.tyBtnAIVAvail1.bValue		:= p_tyDI.bSOT1AIVAvailable;
		tyP0940CommCtrl.tySOT.tyBtnAIVSLarge1.bValue	:= p_tyDI.bSOT1AIVSizeLarge;

		tyP0940CommCtrl.tySOT.tyBtnAIVRcv2.bValue		:= p_tyDI.bSOT2Receive;
		tyP0940CommCtrl.tySOT.tyBtnAIVErr2.bValue		:= p_tyDI.bSOT2AIVError;
		tyP0940CommCtrl.tySOT.tyBtnAIVRdy2.bValue		:= p_tyDI.bSOT2AIVReady;
		tyP0940CommCtrl.tySOT.tyBtnAIVAvail2.bValue		:= p_tyDI.bSOT2AIVAvailable;
		tyP0940CommCtrl.tySOT.tyBtnAIVSLarge2.bValue	:= p_tyDI.bSOT2AIVSizeLarge;

		tyP0940CommCtrl.tySOT.tyBtnAIVRcv3.bValue		:= p_tyDI.bSOT3Receive;
		tyP0940CommCtrl.tySOT.tyBtnAIVErr3.bValue		:= p_tyDI.bSOT3AIVError;
		tyP0940CommCtrl.tySOT.tyBtnAIVRdy3.bValue		:= p_tyDI.bSOT3AIVReady;
		tyP0940CommCtrl.tySOT.tyBtnAIVAvail3.bValue		:= p_tyDI.bSOT3AIVAvailable;
		tyP0940CommCtrl.tySOT.tyBtnAIVSLarge3.bValue	:= p_tyDI.bSOT3AIVSizeLarge;

		tyP0940CommCtrl.tySOT.tyBtnAIVRcv4.bValue		:= p_tyDI.bSOT4Receive;
		tyP0940CommCtrl.tySOT.tyBtnAIVErr4.bValue		:= p_tyDI.bSOT4AIVError;
		tyP0940CommCtrl.tySOT.tyBtnAIVRdy4.bValue		:= p_tyDI.bSOT4AIVReady;
		tyP0940CommCtrl.tySOT.tyBtnAIVAvail4.bValue		:= p_tyDI.bSOT4AIVAvailable;
		tyP0940CommCtrl.tySOT.tyBtnAIVSLarge4.bValue	:= p_tyDI.bSOT4AIVSizeLarge;

		tyP0940CommCtrl.tySOT.tyBtnFleetMgrActive.bValue := p_tyDI.bFleetManagerReady;

	ELSIF p_tyMcParamCurr.eAGVComProtocol = McSetAGVCommOPCUA AND p_tyNtParamCurr.bProjSOTSensorPrep = FALSE THEN

		tyP0940CommCtrl.tySOT.tyBtnAIVErr1.bValue		:= p_tyTagFromMes.tyTagStatOfPlatforms[1].bError;
		tyP0940CommCtrl.tySOT.tyBtnAIVRdy1.bValue		:= p_tyTagFromMes.tyTagStatOfPlatforms[1].bReady;
		tyP0940CommCtrl.tySOT.tyBtnAIVAvail1.bValue		:= p_tyTagFromMes.tyTagStatOfPlatforms[1].bAvailable;
		tyP0940CommCtrl.tySOT.tyBtnAIVSLarge1.bValue	:= p_tyTagFromMes.tyTagStatOfPlatforms[1].bSizeLarge;

		tyP0940CommCtrl.tySOT.tyBtnAIVErr2.bValue		:= p_tyTagFromMes.tyTagStatOfPlatforms[2].bError;
		tyP0940CommCtrl.tySOT.tyBtnAIVRdy2.bValue		:= p_tyTagFromMes.tyTagStatOfPlatforms[2].bReady;
		tyP0940CommCtrl.tySOT.tyBtnAIVAvail2.bValue		:= p_tyTagFromMes.tyTagStatOfPlatforms[2].bAvailable;
		tyP0940CommCtrl.tySOT.tyBtnAIVSLarge2.bValue	:= p_tyTagFromMes.tyTagStatOfPlatforms[2].bSizeLarge;

		tyP0940CommCtrl.tySOT.tyBtnAIVErr3.bValue		:= p_tyTagFromMes.tyTagStatOfPlatforms[3].bError;
		tyP0940CommCtrl.tySOT.tyBtnAIVRdy3.bValue		:= p_tyTagFromMes.tyTagStatOfPlatforms[3].bReady;
		tyP0940CommCtrl.tySOT.tyBtnAIVAvail3.bValue		:= p_tyTagFromMes.tyTagStatOfPlatforms[3].bAvailable;
		tyP0940CommCtrl.tySOT.tyBtnAIVSLarge3.bValue	:= p_tyTagFromMes.tyTagStatOfPlatforms[3].bSizeLarge;

		tyP0940CommCtrl.tySOT.tyBtnAIVErr4.bValue		:= p_tyTagFromMes.tyTagStatOfPlatforms[4].bError;
		tyP0940CommCtrl.tySOT.tyBtnAIVRdy4.bValue		:= p_tyTagFromMes.tyTagStatOfPlatforms[4].bReady;
		tyP0940CommCtrl.tySOT.tyBtnAIVAvail4.bValue		:= p_tyTagFromMes.tyTagStatOfPlatforms[4].bAvailable;
		tyP0940CommCtrl.tySOT.tyBtnAIVSLarge4.bValue	:= p_tyTagFromMes.tyTagStatOfPlatforms[4].bSizeLarge;

		tyP0940CommCtrl.tySOT.tyBtnFleetMgrActive.bValue := p_tyTagFromMes.bActive;
	END_IF

	IF p_tyMcParamCurr.eAGVComProtocol = McSetAGVCommDisabled THEN
		tyP0940CommCtrl.tySOT.tyBtnAIVErr1.bValue		:= FALSE;
		tyP0940CommCtrl.tySOT.tyBtnAIVRdy1.bValue		:= FALSE;
		tyP0940CommCtrl.tySOT.tyBtnAIVAvail1.bValue		:= FALSE;
		tyP0940CommCtrl.tySOT.tyBtnAIVSLarge1.bValue	:= FALSE;

		tyP0940CommCtrl.tySOT.tyBtnAIVErr2.bValue		:= FALSE;
		tyP0940CommCtrl.tySOT.tyBtnAIVRdy2.bValue		:= FALSE;
		tyP0940CommCtrl.tySOT.tyBtnAIVAvail2.bValue		:= FALSE;
		tyP0940CommCtrl.tySOT.tyBtnAIVSLarge2.bValue	:= FALSE;

		tyP0940CommCtrl.tySOT.tyBtnAIVErr3.bValue		:= FALSE;
		tyP0940CommCtrl.tySOT.tyBtnAIVRdy3.bValue		:= FALSE;
		tyP0940CommCtrl.tySOT.tyBtnAIVAvail3.bValue		:= FALSE;
		tyP0940CommCtrl.tySOT.tyBtnAIVSLarge3.bValue	:= FALSE;

		tyP0940CommCtrl.tySOT.tyBtnAIVErr4.bValue		:= FALSE;
		tyP0940CommCtrl.tySOT.tyBtnAIVRdy4.bValue		:= FALSE;
		tyP0940CommCtrl.tySOT.tyBtnAIVAvail4.bValue		:= FALSE;
		tyP0940CommCtrl.tySOT.tyBtnAIVSLarge4.bValue	:= FALSE;

		tyP0940CommCtrl.tySOT.tyBtnFleetMgrActive.bValue := FALSE;
	END_IF

END_ACTION
```

#### Act_OptP0940RstMnl.st
```iecst
ACTION Act_OptP0940RstMnl:

	IF EDGEPOS((bManualMod = FALSE) OR (p_eDSSMEMAAStatus = Error)) THEN
		eDSSMEMAAAct	:= SMEMAActIdle;

		tyP0940CommCtrl.tyDSSMEMAA.tyBtnDBA.bValue	:= FALSE;
	END_IF

	IF EDGEPOS((bManualMod = FALSE) OR (p_eDSSMEMABStatus = Error)) THEN
		eDSSMEMABAct	:= SMEMAActIdle;

		tyP0940CommCtrl.tyDSSMEMAB.tyBtnDBA.bValue	:= FALSE;
	END_IF

	IF EDGEPOS(bManualMod = FALSE) THEN
		tyP0940CommCtrl.tySOT.tyBtnMagErr1.bValue := FALSE;
		tyP0940CommCtrl.tySOT.tyBtnMagErr2.bValue := FALSE;
		tyP0940CommCtrl.tySOT.tyBtnMagErr3.bValue := FALSE;
		tyP0940CommCtrl.tySOT.tyBtnMagErr4.bValue := FALSE;

		tyP0940CommCtrl.tySOT.tyBtnMagRdy1.bValue := FALSE;
		tyP0940CommCtrl.tySOT.tyBtnMagRdy2.bValue := FALSE;
		tyP0940CommCtrl.tySOT.tyBtnMagRdy3.bValue := FALSE;
		tyP0940CommCtrl.tySOT.tyBtnMagRdy4.bValue := FALSE;

		tyP0940CommCtrl.tySOT.tyBtnMagAvail1.bValue := FALSE;
		tyP0940CommCtrl.tySOT.tyBtnMagAvail2.bValue := FALSE;
		tyP0940CommCtrl.tySOT.tyBtnMagAvail3.bValue := FALSE;
		tyP0940CommCtrl.tySOT.tyBtnMagAvail4.bValue := FALSE;

		tyP0940CommCtrl.tySOT.tyBtnMagSLarge1.bValue := FALSE;
		tyP0940CommCtrl.tySOT.tyBtnMagSLarge2.bValue := FALSE;
		tyP0940CommCtrl.tySOT.tyBtnMagSLarge3.bValue := FALSE;
		tyP0940CommCtrl.tySOT.tyBtnMagSLarge4.bValue := FALSE;

		bSOTMagErr1 := FALSE;
		bSOTMagErr2 := FALSE;
		bSOTMagErr3 := FALSE;
		bSOTMagErr4 := FALSE;

		bSOTMagRdy1 := FALSE;
		bSOTMagRdy2 := FALSE;
		bSOTMagRdy3 := FALSE;
		bSOTMagRdy4 := FALSE;

		bSOTMagAvail1 := FALSE;
		bSOTMagAvail2 := FALSE;
		bSOTMagAvail3 := FALSE;
		bSOTMagAvail4 := FALSE;

		bSOTMagSLarge1 := FALSE;
		bSOTMagSLarge2 := FALSE;
		bSOTMagSLarge3 := FALSE;
		bSOTMagSLarge4 := FALSE;

		bAIVReqBring1 := FALSE;
		bAIVReqBring2 := FALSE;
		bAIVReqBring3 := FALSE;
		bAIVReqBring4 := FALSE;

		bAIVReqGet1 := FALSE;
		bAIVReqGet2 := FALSE;
		bAIVReqGet3 := FALSE;
		bAIVReqGet4 := FALSE;

	END_IF

END_ACTION
```

#### Act_OptP0940WriteDO.st
```iecst
ACTION Act_OptP0940WriteDO:

	//DBAA
	IF tyP0940CommCtrl.tyDSSMEMAA.tyBtnDBA.bRtCompl = TRUE THEN
		IF tyP0940CommCtrl.tyDSSMEMAA.tyBtnDBA.bValue = TRUE THEN
			eDSSMEMAAAct	:= SMEMAActSetSig;

			IF p_eDSSMEMAAStat = SMEMAActSetSig AND p_eDSSMEMAAStatus = Done THEN
				eDSSMEMAAAct	:= SMEMAActIdle;

				tyP0940CommCtrl.tyDSSMEMAA.tyBtnDBA.bRtCompl	:= FALSE;
			END_IF

		ELSE
			eDSSMEMAAAct	:= SMEMAActRstSig;

			IF p_eDSSMEMAAStat = SMEMAActRstSig AND p_eDSSMEMAAStatus = Done THEN
				eDSSMEMAAAct	:= SMEMAActIdle;

				tyP0940CommCtrl.tyDSSMEMAA.tyBtnDBA.bRtCompl	:= FALSE;
			END_IF

		END_IF

	END_IF

	//DBAB
	IF tyP0940CommCtrl.tyDSSMEMAB.tyBtnDBA.bRtCompl = TRUE THEN
		IF tyP0940CommCtrl.tyDSSMEMAB.tyBtnDBA.bValue = TRUE THEN
			eDSSMEMABAct	:= SMEMAActSetSig;

			IF p_eDSSMEMABStat = SMEMAActSetSig AND p_eDSSMEMABStatus = Done THEN
				eDSSMEMABAct	:= SMEMAActIdle;

				tyP0940CommCtrl.tyDSSMEMAB.tyBtnDBA.bRtCompl	:= FALSE;
			END_IF

		ELSE
			eDSSMEMABAct	:= SMEMAActRstSig;

			IF p_eDSSMEMABStat = SMEMAActRstSig AND p_eDSSMEMABStatus = Done THEN
				eDSSMEMABAct	:= SMEMAActIdle;

				tyP0940CommCtrl.tyDSSMEMAB.tyBtnDBA.bRtCompl	:= FALSE;
			END_IF

		END_IF

	END_IF

	IF p_tyMcParamCurr.eAGVComProtocol <> McSetAGVCommDisabled THEN
		//Error
		IF tyP0940CommCtrl.tySOT.tyBtnMagErr1.bRtCompl = TRUE THEN

			IF tyP0940CommCtrl.tySOT.tyBtnMagErr1.bValue = TRUE THEN
				bSOTMagErr1 := TRUE;
				tyP0940CommCtrl.tySOT.tyBtnMagErr1.bRtCompl := FALSE;
			ELSE
				bSOTMagErr1 := FALSE;
				tyP0940CommCtrl.tySOT.tyBtnMagErr1.bRtCompl := FALSE;
			END_IF
		END_IF

		IF tyP0940CommCtrl.tySOT.tyBtnMagErr2.bRtCompl = TRUE THEN

			IF tyP0940CommCtrl.tySOT.tyBtnMagErr2.bValue = TRUE THEN
				bSOTMagErr2 := TRUE;
				tyP0940CommCtrl.tySOT.tyBtnMagErr2.bRtCompl := FALSE;
			ELSE
				bSOTMagErr2 := FALSE;
				tyP0940CommCtrl.tySOT.tyBtnMagErr2.bRtCompl := FALSE;
			END_IF
		END_IF

		IF tyP0940CommCtrl.tySOT.tyBtnMagErr3.bRtCompl = TRUE THEN

			IF tyP0940CommCtrl.tySOT.tyBtnMagErr3.bValue = TRUE THEN
				bSOTMagErr3 := TRUE;
				tyP0940CommCtrl.tySOT.tyBtnMagErr3.bRtCompl := FALSE;
			ELSE
				bSOTMagErr3 := FALSE;
				tyP0940CommCtrl.tySOT.tyBtnMagErr3.bRtCompl := FALSE;
			END_IF
		END_IF

		IF tyP0940CommCtrl.tySOT.tyBtnMagErr4.bRtCompl = TRUE THEN

			IF tyP0940CommCtrl.tySOT.tyBtnMagErr4.bValue = TRUE THEN
				bSOTMagErr4 := TRUE;
				tyP0940CommCtrl.tySOT.tyBtnMagErr4.bRtCompl := FALSE;
			ELSE
				bSOTMagErr4 := FALSE;
				tyP0940CommCtrl.tySOT.tyBtnMagErr4.bRtCompl := FALSE;
			END_IF
		END_IF

		//Ready
		IF tyP0940CommCtrl.tySOT.tyBtnMagRdy1.bRtCompl = TRUE THEN

			IF tyP0940CommCtrl.tySOT.tyBtnMagRdy1.bValue = TRUE THEN
				bSOTMagRdy1 := TRUE;
				tyP0940CommCtrl.tySOT.tyBtnMagRdy1.bRtCompl := FALSE;
			ELSE
				bSOTMagRdy1 := FALSE;
				tyP0940CommCtrl.tySOT.tyBtnMagRdy1.bRtCompl := FALSE;
			END_IF
		END_IF

		IF tyP0940CommCtrl.tySOT.tyBtnMagRdy2.bRtCompl = TRUE THEN

			IF tyP0940CommCtrl.tySOT.tyBtnMagRdy2.bValue = TRUE THEN
				bSOTMagRdy2 := TRUE;
				tyP0940CommCtrl.tySOT.tyBtnMagRdy2.bRtCompl := FALSE;
			ELSE
				bSOTMagRdy2 := FALSE;
				tyP0940CommCtrl.tySOT.tyBtnMagRdy2.bRtCompl := FALSE;
			END_IF
		END_IF

		IF tyP0940CommCtrl.tySOT.tyBtnMagRdy3.bRtCompl = TRUE THEN

			IF tyP0940CommCtrl.tySOT.tyBtnMagRdy3.bValue = TRUE THEN
				bSOTMagRdy3 := TRUE;
				tyP0940CommCtrl.tySOT.tyBtnMagRdy3.bRtCompl := FALSE;
			ELSE
				bSOTMagRdy3 := FALSE;
				tyP0940CommCtrl.tySOT.tyBtnMagRdy3.bRtCompl := FALSE;
			END_IF
		END_IF

		IF tyP0940CommCtrl.tySOT.tyBtnMagRdy4.bRtCompl = TRUE THEN

			IF tyP0940CommCtrl.tySOT.tyBtnMagRdy4.bValue = TRUE THEN
				bSOTMagRdy4 := TRUE;
				tyP0940CommCtrl.tySOT.tyBtnMagRdy4.bRtCompl := FALSE;
			ELSE
				bSOTMagRdy4 := FALSE;
				tyP0940CommCtrl.tySOT.tyBtnMagRdy4.bRtCompl := FALSE;
			END_IF
		END_IF

		//Available
		IF tyP0940CommCtrl.tySOT.tyBtnMagAvail1.bRtCompl = TRUE THEN

			IF tyP0940CommCtrl.tySOT.tyBtnMagAvail1.bValue = TRUE THEN
				bSOTMagAvail1 := TRUE;
				tyP0940CommCtrl.tySOT.tyBtnMagAvail1.bRtCompl := FALSE;
			ELSE
				bSOTMagAvail1 := FALSE;
				tyP0940CommCtrl.tySOT.tyBtnMagAvail1.bRtCompl := FALSE;
			END_IF
		END_IF

		IF tyP0940CommCtrl.tySOT.tyBtnMagAvail2.bRtCompl = TRUE THEN

			IF tyP0940CommCtrl.tySOT.tyBtnMagAvail2.bValue = TRUE THEN
				bSOTMagAvail2 := TRUE;
				tyP0940CommCtrl.tySOT.tyBtnMagAvail2.bRtCompl := FALSE;
			ELSE
				bSOTMagAvail2 := FALSE;
				tyP0940CommCtrl.tySOT.tyBtnMagAvail2.bRtCompl := FALSE;
			END_IF
		END_IF

		IF tyP0940CommCtrl.tySOT.tyBtnMagAvail3.bRtCompl = TRUE THEN

			IF tyP0940CommCtrl.tySOT.tyBtnMagAvail3.bValue = TRUE THEN
				bSOTMagAvail3 := TRUE;
				tyP0940CommCtrl.tySOT.tyBtnMagAvail3.bRtCompl := FALSE;
			ELSE
				bSOTMagAvail3 := FALSE;
				tyP0940CommCtrl.tySOT.tyBtnMagAvail3.bRtCompl := FALSE;
			END_IF
		END_IF

		IF tyP0940CommCtrl.tySOT.tyBtnMagAvail4.bRtCompl = TRUE THEN

			IF tyP0940CommCtrl.tySOT.tyBtnMagAvail4.bValue = TRUE THEN
				bSOTMagAvail4 := TRUE;
				tyP0940CommCtrl.tySOT.tyBtnMagAvail4.bRtCompl := FALSE;
			ELSE
				bSOTMagAvail4 := FALSE;
				tyP0940CommCtrl.tySOT.tyBtnMagAvail4.bRtCompl := FALSE;
			END_IF
		END_IF

		//Size
		IF tyP0940CommCtrl.tySOT.tyBtnMagSLarge1.bRtCompl = TRUE THEN

			IF tyP0940CommCtrl.tySOT.tyBtnMagSLarge1.bValue = TRUE THEN
				bSOTMagSLarge1 := TRUE;
				tyP0940CommCtrl.tySOT.tyBtnMagSLarge1.bRtCompl := FALSE;
			ELSE
				bSOTMagSLarge1 := FALSE;
				tyP0940CommCtrl.tySOT.tyBtnMagSLarge1.bRtCompl := FALSE;
			END_IF
		END_IF

		IF tyP0940CommCtrl.tySOT.tyBtnMagSLarge2.bRtCompl = TRUE THEN

			IF tyP0940CommCtrl.tySOT.tyBtnMagSLarge2.bValue = TRUE THEN
				bSOTMagSLarge2 := TRUE;
				tyP0940CommCtrl.tySOT.tyBtnMagSLarge2.bRtCompl := FALSE;
			ELSE
				bSOTMagSLarge2 := FALSE;
				tyP0940CommCtrl.tySOT.tyBtnMagSLarge2.bRtCompl := FALSE;
			END_IF
		END_IF

		IF tyP0940CommCtrl.tySOT.tyBtnMagSLarge3.bRtCompl = TRUE THEN

			IF tyP0940CommCtrl.tySOT.tyBtnMagSLarge3.bValue = TRUE THEN
				bSOTMagSLarge3 := TRUE;
				tyP0940CommCtrl.tySOT.tyBtnMagSLarge3.bRtCompl := FALSE;
			ELSE
				bSOTMagSLarge3 := FALSE;
				tyP0940CommCtrl.tySOT.tyBtnMagSLarge3.bRtCompl := FALSE;
			END_IF
		END_IF

		IF tyP0940CommCtrl.tySOT.tyBtnMagSLarge4.bRtCompl = TRUE THEN

			IF tyP0940CommCtrl.tySOT.tyBtnMagSLarge4.bValue = TRUE THEN
				bSOTMagSLarge4 := TRUE;
				tyP0940CommCtrl.tySOT.tyBtnMagSLarge4.bRtCompl := FALSE;
			ELSE
				bSOTMagSLarge4 := FALSE;
				tyP0940CommCtrl.tySOT.tyBtnMagSLarge4.bRtCompl := FALSE;
			END_IF
		END_IF

		//Req Bring
		IF tyP0940CommCtrl.tySOT.tyBtnMagReqBring1.bRtCompl = TRUE THEN

			IF tyP0940CommCtrl.tySOT.tyBtnMagReqBring1.bValue = TRUE THEN
				bAIVReqBring1 := TRUE;
				tyP0940CommCtrl.tySOT.tyBtnMagReqBring1.bRtCompl := FALSE;
			ELSE
				bAIVReqBring1 := FALSE;
				tyP0940CommCtrl.tySOT.tyBtnMagReqBring1.bRtCompl := FALSE;
			END_IF
		END_IF

		IF tyP0940CommCtrl.tySOT.tyBtnMagReqBring2.bRtCompl = TRUE THEN

			IF tyP0940CommCtrl.tySOT.tyBtnMagReqBring2.bValue = TRUE THEN
				bAIVReqBring2 := TRUE;
				tyP0940CommCtrl.tySOT.tyBtnMagReqBring2.bRtCompl := FALSE;
			ELSE
				bAIVReqBring2 := FALSE;
				tyP0940CommCtrl.tySOT.tyBtnMagReqBring2.bRtCompl := FALSE;
			END_IF
		END_IF

		IF tyP0940CommCtrl.tySOT.tyBtnMagReqBring3.bRtCompl = TRUE THEN

			IF tyP0940CommCtrl.tySOT.tyBtnMagReqBring3.bValue = TRUE THEN
				bAIVReqBring1 := TRUE;
				tyP0940CommCtrl.tySOT.tyBtnMagReqBring3.bRtCompl := FALSE;
			ELSE
				bAIVReqBring1 := FALSE;
				tyP0940CommCtrl.tySOT.tyBtnMagReqBring3.bRtCompl := FALSE;
			END_IF
		END_IF

		IF tyP0940CommCtrl.tySOT.tyBtnMagReqBring4.bRtCompl = TRUE THEN

			IF tyP0940CommCtrl.tySOT.tyBtnMagReqBring4.bValue = TRUE THEN
				bAIVReqBring1 := TRUE;
				tyP0940CommCtrl.tySOT.tyBtnMagReqBring4.bRtCompl := FALSE;
			ELSE
				bAIVReqBring1 := FALSE;
				tyP0940CommCtrl.tySOT.tyBtnMagReqBring4.bRtCompl := FALSE;
			END_IF
		END_IF

		//Req Get
		IF tyP0940CommCtrl.tySOT.tyBtnMagReqtGet1.bRtCompl = TRUE THEN

			IF tyP0940CommCtrl.tySOT.tyBtnMagReqtGet1.bValue = TRUE THEN
				bAIVReqGet1 := TRUE;
				tyP0940CommCtrl.tySOT.tyBtnMagReqtGet1.bRtCompl := FALSE;
			ELSE
				bAIVReqGet1 := FALSE;
				tyP0940CommCtrl.tySOT.tyBtnMagReqtGet1.bRtCompl := FALSE;
			END_IF
		END_IF

		IF tyP0940CommCtrl.tySOT.tyBtnMagReqtGet2.bRtCompl = TRUE THEN

			IF tyP0940CommCtrl.tySOT.tyBtnMagReqtGet2.bValue = TRUE THEN
				bAIVReqGet2 := TRUE;
				tyP0940CommCtrl.tySOT.tyBtnMagReqtGet2.bRtCompl := FALSE;
			ELSE
				bAIVReqGet2 := FALSE;
				tyP0940CommCtrl.tySOT.tyBtnMagReqtGet2.bRtCompl := FALSE;
			END_IF
		END_IF

		IF tyP0940CommCtrl.tySOT.tyBtnMagReqtGet3.bRtCompl = TRUE THEN

			IF tyP0940CommCtrl.tySOT.tyBtnMagReqtGet3.bValue = TRUE THEN
				bAIVReqGet3 := TRUE;
				tyP0940CommCtrl.tySOT.tyBtnMagReqtGet3.bRtCompl := FALSE;
			ELSE
				bAIVReqGet3 := FALSE;
				tyP0940CommCtrl.tySOT.tyBtnMagReqtGet3.bRtCompl := FALSE;
			END_IF
		END_IF

		IF tyP0940CommCtrl.tySOT.tyBtnMagReqtGet4.bRtCompl = TRUE THEN

			IF tyP0940CommCtrl.tySOT.tyBtnMagReqtGet4.bValue = TRUE THEN
				bAIVReqGet4 := TRUE;
				tyP0940CommCtrl.tySOT.tyBtnMagReqtGet4.bRtCompl := FALSE;
			ELSE
				bAIVReqGet4 := FALSE;
				tyP0940CommCtrl.tySOT.tyBtnMagReqtGet4.bRtCompl := FALSE;
			END_IF
		END_IF
	END_IF

END_ACTION
```

#### Act_EntP0950Disp.st
```iecst
ACTION Act_EntP0950Disp:

	// Access Address
	p_tyC0002FullMask ACCESS ADR (tyP0950Simu.tyFullMaskHide);

	p_tyC0005Main ACCESS ADR(tyCommon.tyMain);

	p_tyC0007Notif ACCESS ADR(tyCommon.tyNotif);

	p_tyC0009Info ACCESS ADR(tyCommon.tyInfo);

	p_tyP0950Simu ACCESS ADR(tyP0950Simu.tySimu);

	p_tyP0950SimuAGVtoMC ACCESS ADR(tyP0950Simu.tyAGVToMc);
	p_tyP0950SimuMCtoAGV ACCESS ADR(tyP0950Simu.tyMcToAGV);

	//Display
	tyP0950Simu.tyAGVToMc.tyLyr.uiRtStat.0 := NOT(p_tyNtParamCurr.bProjAGVPrep AND p_tyMcParamCurr.bAGVComEn);

END_ACTION
```
